   Verteiler_O2.Values[106] := 0.0;
   Verteiler_O2.Values[107] := 0.0;
   Verteiler_O2.Values[108] := 0.0;
   Verteiler_O2.Values[109] := 0.0;
   Verteiler_O2.Values[110] := 0.0;
   Verteiler_O2.Values[111] := 0.0;
   Verteiler_O2.Values[112] := 0.0;
   Verteiler_O2.Values[113] := 0.0;
   Verteiler_O2.Values[114] := 0.0;
   Verteiler_O2.Values[115] := 0.0;
   Verteiler_O2.Values[116] := 0.0;
   Verteiler_O2.Values[117] := 0.0;
   Verteiler_O2.Values[118] := 0.0;
   Verteiler_O2.Values[119] := 0.0;
   Verteiler_Temp.Values[0] := 0.0;
   Verteiler_Temp.Values[1] := 0.0;
   Verteiler_Temp.Values[2] := 0.0;
   Verteiler_Temp.Values[3] := 0.0;
   Verteiler_Temp.Values[4] := 0.0;
   Verteiler_Temp.Values[5] := 0.0;
   Verteiler_Temp.Values[6] := 0.0;
   Verteiler_Temp.Values[7] := 0.0;
   Verteiler_Temp.Values[8] := 0.0;
   Verteiler_Temp.Values[9] := 0.0;
   Verteiler_Temp.Values[10] := 0.0;
   Verteiler_Temp.Values[11] := 0.0;
   Verteiler_Temp.Values[12] := 0.0;
   Verteiler_Temp.Values[13] := 0.0;
   Verteiler_Temp.Values[14] := 0.0;
   Verteiler_Temp.Values[15] := 0.0;
   Verteiler_Temp.Values[16] := 0.0;
   Verteiler_Temp.Values[17] := 0.0;
   Verteiler_Temp.Values[18] := 0.0;
   Verteiler_Temp.Values[19] := 0.0;
   Verteiler_Temp.Values[20] := 0.0;
   Verteiler_Temp.Values[21] := 0.0;
   Verteiler_Temp.Values[22] := 0.0;
   Verteiler_Temp.Values[23] := 0.0;
   Verteiler_Temp.Values[24] := 0.0;
   Verteiler_Temp.Values[25] := 0.0;
   Verteiler_Temp.Values[26] := 0.0;
   Verteiler_Temp.Values[27] := 0.0;
   Verteiler_Temp.Values[28] := 0.0;
   Verteiler_Temp.Values[29] := 0.0;
   Verteiler_Temp.Values[30] := 0.0;
   Verteiler_Temp.Values[31] := 0.0;
   Verteiler_Temp.Values[32] := 0.0;
   Verteiler_Temp.Values[33] := 0.0;
   Verteiler_Temp.Values[34] := 0.0;
   Verteiler_Temp.Values[35] := 0.0;
   Verteiler_Temp.Values[36] := 0.0;
   Verteiler_Temp.Values[37] := 0.0;
   Verteiler_Temp.Values[38] := 0.0;
   Verteiler_Temp.Values[39] := 0.0;
   Verteiler_Temp.Values[40] := 0.0;
   Verteiler_Temp.Values[41] := 0.0;
   Verteiler_Temp.Values[42] := 0.0;
   Verteiler_Temp.Values[43] := 0.0;
   Verteiler_Temp.Values[44] := 0.0;
   Verteiler_Temp.Values[45] := 0.0;
   Verteiler_Temp.Values[46] := 0.0;
   Verteiler_Temp.Values[47] := 0.0;
   Verteiler_Temp.Values[48] := 0.0;
   Verteiler_Temp.Values[49] := 0.0;
   Verteiler_Temp.Values[50] := 0.0;
   Verteiler_Temp.Values[51] := 0.0;
   Verteiler_Temp.Values[52] := 0.0;
   Verteiler_Temp.Values[53] := 0.0;
   Verteiler_Temp.Values[54] := 0.0;
   Verteiler_Temp.Values[55] := 0.0;
   Verteiler_Temp.Values[56] := 0.0;
   Verteiler_Temp.Values[57] := 0.0;
   Verteiler_Temp.Values[58] := 0.0;
   Verteiler_Temp.Values[59] := 0.0;
   Verteiler_Temp.Values[60] := 0.0;
   Verteiler_Temp.Values[61] := 0.0;
   Verteiler_Temp.Values[62] := 0.0;
   Verteiler_Temp.Values[63] := 0.0;
   Verteiler_Temp.Values[64] := 0.0;
   Verteiler_Temp.Values[65] := 0.0;
   Verteiler_Temp.Values[66] := 0.0;
   Verteiler_Temp.Values[67] := 0.0;
   Verteiler_Temp.Values[68] := 0.0;
   Verteiler_Temp.Values[69] := 0.0;
   Verteiler_Temp.Values[70] := 0.0;
   Verteiler_Temp.Values[71] := 0.0;
   Verteiler_Temp.Values[72] := 0.0;
   Verteiler_Temp.Values[73] := 0.0;
   Verteiler_Temp.Values[74] := 0.0;
   Verteiler_Temp.Values[75] := 0.0;
   Verteiler_Temp.Values[76] := 0.0;
   Verteiler_Temp.Values[77] := 0.0;
   Verteiler_Temp.Values[78] := 0.0;
   Verteiler_Temp.Values[79] := 0.0;
   Verteiler_Temp.Values[80] := 0.0;
   Verteiler_Temp.Values[81] := 0.0;
   Verteiler_Temp.Values[82] := 0.0;
   Verteiler_Temp.Values[83] := 0.0;
   Verteiler_Temp.Values[84] := 0.0;
   Verteiler_Temp.Values[85] := 0.0;
   Verteiler_Temp.Values[86] := 0.0;
   Verteiler_Temp.Values[87] := 0.0;
   Verteiler_Temp.Values[88] := 0.0;
   Verteiler_Temp.Values[89] := 0.0;
   Verteiler_Temp.Values[90] := 0.0;
   Verteiler_Temp.Values[91] := 0.0;
   Verteiler_Temp.Values[92] := 0.0;
   Verteiler_Temp.Values[93] := 0.0;
   Verteiler_Temp.Values[94] := 0.0;
   Verteiler_Temp.Values[95] := 0.0;
   Verteiler_Temp.Values[96] := 0.0;
   Verteiler_Temp.Values[97] := 0.0;
   Verteiler_Temp.Values[98] := 0.0;
   Verteiler_Temp.Values[99] := 0.0;
   Verteiler_Temp.Values[100] := 0.0;
   Verteiler_Temp.Values[101] := 0.0;
   Verteiler_Temp.Values[102] := 0.0;
   Verteiler_Temp.Values[103] := 0.0;
   Verteiler_Temp.Values[104] := 0.0;
   Verteiler_Temp.Values[105] := 0.0;
   Verteiler_Temp.Values[106] := 0.0;
   Verteiler_Temp.Values[107] := 0.0;
   Verteiler_Temp.Values[108] := 0.0;
   Verteiler_Temp.Values[109] := 0.0;
   Verteiler_Temp.Values[110] := 0.0;
   Verteiler_Temp.Values[111] := 0.0;
   Verteiler_Temp.Values[112] := 0.0;
   Verteiler_Temp.Values[113] := 0.0;
   Verteiler_Temp.Values[114] := 0.0;
   Verteiler_Temp.Values[115] := 0.0;
   Verteiler_Temp.Values[116] := 0.0;
   Verteiler_Temp.Values[117] := 0.0;
   Verteiler_Temp.Values[118] := 0.0;
   Verteiler_Temp.Values[119] := 0.0;
   BB_UeSS_DF.Values[0] := -0.0063294;
   BB_UeSS_DF.Values[1] := -0.0063294;
   BB_UeSS_DF.Values[2] := -0.0063294;
   BB_UeSS_DF.Values[3] := -0.0063294;
   BB_UeSS_DF.Values[4] := -0.0063294;
   BB_UeSS_DF.Values[5] := -0.0063294;
   BB_UeSS_DF.Values[6] := -0.0063294;
   BB_UeSS_DF.Values[7] := -0.0063294;
   BB_UeSS_DF.Values[8] := -0.0099462;
   BB_UeSS_DF.Values[9] := -0.009042;
   BB_UeSS_DF.Values[10] := 0.0;
   BB_UeSS_DF.Values[11] := 0.0;
   BB_UeSS_DF.Values[12] := 0.0;
   BB_UeSS_DF.Values[13] := 0.0;
   BB_UeSS_DF.Values[14] := 0.0;
   BB_UeSS_DF.Values[15] := 0.0;
   BB_UeSS_DF.Values[16] := 0.0;
   BB_UeSS_DF.Values[17] := 0.0;
   BB_UeSS_DF.Values[18] := 0.0;
   BB_UeSS_DF.Values[19] := 0.0;
   BB_UeSS_DF.Values[20] := 0.0;
   BB_UeSS_DF.Values[21] := 0.0;
   BB_UeSS_DF.Values[22] := 0.0;
   BB_UeSS_DF.Values[23] := 0.0;
   BB_UeSS_DF.Values[24] := 0.0;
   BB_UeSS_DF.Values[25] := 0.0;
   BB_UeSS_DF.Values[26] := 0.0;
   BB_UeSS_DF.Values[27] := 0.0;
   BB_UeSS_DF.Values[28] := 0.0;
   BB_UeSS_DF.Values[29] := 0.0;
   BB_UeSS_DF.Values[30] := 0.0;
   BB_UeSS_DF.Values[31] := 0.0;
   BB_UeSS_DF.Values[32] := 0.0;
   BB_UeSS_DF.Values[33] := 0.0;
   BB_UeSS_DF.Values[34] := 0.0;
   BB_UeSS_DF.Values[35] := 0.0;
   BB_UeSS_DF.Values[36] := 0.0;
   BB_UeSS_DF.Values[37] := 0.0;
   BB_UeSS_DF.Values[38] := 0.0;
   BB_UeSS_DF.Values[39] := 0.0;
   BB_UeSS_DF.Values[40] := 0.0;
   BB_UeSS_DF.Values[41] := 0.0;
   BB_UeSS_DF.Values[42] := 0.0;
   BB_UeSS_DF.Values[43] := 0.0;
   BB_UeSS_DF.Values[44] := 0.0;
   BB_UeSS_DF.Values[45] := 0.0;
   BB_UeSS_DF.Values[46] := 0.0;
   BB_UeSS_DF.Values[47] := 0.0;
   BB_UeSS_DF.Values[48] := 0.0;
   BB_UeSS_DF.Values[49] := 0.0;
   BB_UeSS_DF.Values[50] := 0.0;
   BB_UeSS_DF.Values[51] := 0.0;
   BB_UeSS_DF.Values[52] := 0.0;
   BB_UeSS_DF.Values[53] := 0.0;
   BB_UeSS_DF.Values[54] := 0.0;
   BB_UeSS_DF.Values[55] := 0.0;
   BB_UeSS_DF.Values[56] := 0.0;
   BB_UeSS_DF.Values[57] := 0.0;
   BB_UeSS_DF.Values[58] := 0.0;
   BB_UeSS_DF.Values[59] := 0.0;
   BB_UeSS_DF.Values[60] := 0.0;
   BB_UeSS_DF.Values[61] := 0.0;
   BB_UeSS_DF.Values[62] := 0.0;
   BB_UeSS_DF.Values[63] := 0.0;
   BB_UeSS_DF.Values[64] := 0.0;
   BB_UeSS_DF.Values[65] := 0.0;
   BB_UeSS_DF.Values[66] := 0.0;
   BB_UeSS_DF.Values[67] := 0.0;
   BB_UeSS_DF.Values[68] := 0.0;
   BB_UeSS_DF.Values[69] := 0.0;
   BB_UeSS_DF.Values[70] := 0.0;
   BB_UeSS_DF.Values[71] := 0.0;
   BB_UeSS_DF.Values[72] := 0.0;
   BB_UeSS_DF.Values[73] := 0.0;
   BB_UeSS_DF.Values[74] := 0.0;
   BB_UeSS_DF.Values[75] := 0.0;
   BB_UeSS_DF.Values[76] := 0.0;
   BB_UeSS_DF.Values[77] := 0.0;
   BB_UeSS_DF.Values[78] := 0.0;
   BB_UeSS_DF.Values[79] := 0.0;
   BB_UeSS_DF.Values[80] := 0.0;
   BB_UeSS_DF.Values[81] := 0.0;
   BB_UeSS_DF.Values[82] := 0.0;
   BB_UeSS_DF.Values[83] := 0.0;
   BB_UeSS_DF.Values[84] := 0.0;
   BB_UeSS_DF.Values[85] := 0.0;
   BB_UeSS_DF.Values[86] := 0.0;
   BB_UeSS_DF.Values[87] := 0.0;
   BB_UeSS_DF.Values[88] := 0.0;
   BB_UeSS_DF.Values[89] := 0.0;
   BB_UeSS_DF.Values[90] := 0.0;
   BB_UeSS_DF.Values[91] := 0.0;
   BB_UeSS_DF.Values[92] := 0.0;
   BB_UeSS_DF.Values[93] := 0.0;
   BB_UeSS_DF.Values[94] := 0.0;
   BB_UeSS_DF.Values[95] := 0.0;
   BB_UeSS_DF.Values[96] := 0.0;
   BB_UeSS_DF.Values[97] := 0.0;
   BB_UeSS_DF.Values[98] := 0.0;
   BB_UeSS_DF.Values[99] := 0.0;
   BB_UeSS_DF.Values[100] := 0.0;
   BB_UeSS_DF.Values[101] := 0.0;
   BB_UeSS_DF.Values[102] := 0.0;
   BB_UeSS_DF.Values[103] := 0.0;
   BB_UeSS_DF.Values[104] := 0.0;
   BB_UeSS_DF.Values[105] := 0.0;
   BB_UeSS_DF.Values[106] := 0.0;
   BB_UeSS_DF.Values[107] := 0.0;
   BB_UeSS_DF.Values[108] := 0.0;
   BB_UeSS_DF.Values[109] := 0.0;
   BB_UeSS_DF.Values[110] := 0.0;
   BB_UeSS_DF.Values[111] := 0.0;
   BB_UeSS_DF.Values[112] := 0.0;
   BB_UeSS_DF.Values[113] := 0.0;
   BB_UeSS_DF.Values[114] := 0.0;
   BB_UeSS_DF.Values[115] := 0.0;
   BB_UeSS_DF.Values[116] := 0.0;
   BB_UeSS_DF.Values[117] := 0.0;
   BB_UeSS_DF.Values[118] := 0.0;
   BB_UeSS_DF.Values[119] := 0.0;
   Ablauf_DF.Values[0] := 11.22745;
   Ablauf_DF.Values[1] := 11.21796;
   Ablauf_DF.Values[2] := 11.20439;
   Ablauf_DF.Values[3] := 11.19897;
   Ablauf_DF.Values[4] := 11.18948;
   Ablauf_DF.Values[5] := 11.18541;
   Ablauf_DF.Values[6] := 11.1949;
   Ablauf_DF.Values[7] := 11.22338;
   Ablauf_DF.Values[8] := 11.2383;
   Ablauf_DF.Values[9] := 11.22745;
   Ablauf_DF.Values[10] := 0.0;
   Ablauf_DF.Values[11] := 0.0;
   Ablauf_DF.Values[12] := 0.0;
   Ablauf_DF.Values[13] := 0.0;
   Ablauf_DF.Values[14] := 0.0;
   Ablauf_DF.Values[15] := 0.0;
   Ablauf_DF.Values[16] := 0.0;
   Ablauf_DF.Values[17] := 0.0;
   Ablauf_DF.Values[18] := 0.0;
   Ablauf_DF.Values[19] := 0.0;
   Ablauf_DF.Values[20] := 0.0;
   Ablauf_DF.Values[21] := 0.0;
   Ablauf_DF.Values[22] := 0.0;
   Ablauf_DF.Values[23] := 0.0;
   Ablauf_DF.Values[24] := 0.0;
   Ablauf_DF.Values[25] := 0.0;
   Ablauf_DF.Values[26] := 0.0;
   Ablauf_DF.Values[27] := 0.0;
   Ablauf_DF.Values[28] := 0.0;
   Ablauf_DF.Values[29] := 0.0;
   Ablauf_DF.Values[30] := 0.0;
   Ablauf_DF.Values[31] := 0.0;
   Ablauf_DF.Values[32] := 0.0;
   Ablauf_DF.Values[33] := 0.0;
   Ablauf_DF.Values[34] := 0.0;
   Ablauf_DF.Values[35] := 0.0;
   Ablauf_DF.Values[36] := 0.0;
   Ablauf_DF.Values[37] := 0.0;
   Ablauf_DF.Values[38] := 0.0;
   Ablauf_DF.Values[39] := 0.0;
   Ablauf_DF.Values[40] := 0.0;
   Ablauf_DF.Values[41] := 0.0;
   Ablauf_DF.Values[42] := 0.0;
   Ablauf_DF.Values[43] := 0.0;
   Ablauf_DF.Values[44] := 0.0;
   Ablauf_DF.Values[45] := 0.0;
   Ablauf_DF.Values[46] := 0.0;
   Ablauf_DF.Values[47] := 0.0;
   Ablauf_DF.Values[48] := 0.0;
   Ablauf_DF.Values[49] := 0.0;
   Ablauf_DF.Values[50] := 0.0;
   Ablauf_DF.Values[51] := 0.0;
   Ablauf_DF.Values[52] := 0.0;
   Ablauf_DF.Values[53] := 0.0;
   Ablauf_DF.Values[54] := 0.0;
   Ablauf_DF.Values[55] := 0.0;
   Ablauf_DF.Values[56] := 0.0;
   Ablauf_DF.Values[57] := 0.0;
   Ablauf_DF.Values[58] := 0.0;
   Ablauf_DF.Values[59] := 0.0;
   Ablauf_DF.Values[60] := 0.0;
   Ablauf_DF.Values[61] := 0.0;
   Ablauf_DF.Values[62] := 0.0;
   Ablauf_DF.Values[63] := 0.0;
   Ablauf_DF.Values[64] := 0.0;
   Ablauf_DF.Values[65] := 0.0;
   Ablauf_DF.Values[66] := 0.0;
   Ablauf_DF.Values[67] := 0.0;
   Ablauf_DF.Values[68] := 0.0;
   Ablauf_DF.Values[69] := 0.0;
   Ablauf_DF.Values[70] := 0.0;
   Ablauf_DF.Values[71] := 0.0;
   Ablauf_DF.Values[72] := 0.0;
   Ablauf_DF.Values[73] := 0.0;
   Ablauf_DF.Values[74] := 0.0;
   Ablauf_DF.Values[75] := 0.0;
   Ablauf_DF.Values[76] := 0.0;
   Ablauf_DF.Values[77] := 0.0;
   Ablauf_DF.Values[78] := 0.0;
   Ablauf_DF.Values[79] := 0.0;
   Ablauf_DF.Values[80] := 0.0;
   Ablauf_DF.Values[81] := 0.0;
   Ablauf_DF.Values[82] := 0.0;
   Ablauf_DF.Values[83] := 0.0;
   Ablauf_DF.Values[84] := 0.0;
   Ablauf_DF.Values[85] := 0.0;
   Ablauf_DF.Values[86] := 0.0;
   Ablauf_DF.Values[87] := 0.0;
   Ablauf_DF.Values[88] := 0.0;
   Ablauf_DF.Values[89] := 0.0;
   Ablauf_DF.Values[90] := 0.0;
   Ablauf_DF.Values[91] := 0.0;
   Ablauf_DF.Values[92] := 0.0;
   Ablauf_DF.Values[93] := 0.0;
   Ablauf_DF.Values[94] := 0.0;
   Ablauf_DF.Values[95] := 0.0;
   Ablauf_DF.Values[96] := 0.0;
   Ablauf_DF.Values[97] := 0.0;
   Ablauf_DF.Values[98] := 0.0;
   Ablauf_DF.Values[99] := 0.0;
   Ablauf_DF.Values[100] := 0.0;
   Ablauf_DF.Values[101] := 0.0;
   Ablauf_DF.Values[102] := 0.0;
   Ablauf_DF.Values[103] := 0.0;
   Ablauf_DF.Values[104] := 0.0;
   Ablauf_DF.Values[105] := 0.0;
   Ablauf_DF.Values[106] := 0.0;
   Ablauf_DF.Values[107] := 0.0;
   Ablauf_DF.Values[108] := 0.0;
   Ablauf_DF.Values[109] := 0.0;
   Ablauf_DF.Values[110] := 0.0;
   Ablauf_DF.Values[111] := 0.0;
   Ablauf_DF.Values[112] := 0.0;
   Ablauf_DF.Values[113] := 0.0;
   Ablauf_DF.Values[114] := 0.0;
   Ablauf_DF.Values[115] := 0.0;
   Ablauf_DF.Values[116] := 0.0;
   Ablauf_DF.Values[117] := 0.0;
   Ablauf_DF.Values[118] := 0.0;
   Ablauf_DF.Values[119] := 0.0;
   Ablauf_pH.Values[0] := 7.047787;
   Ablauf_pH.Values[1] := 7.047787;
   Ablauf_pH.Values[2] := 7.047787;
   Ablauf_pH.Values[3] := 7.047787;
   Ablauf_pH.Values[4] := 7.047787;
   Ablauf_pH.Values[5] := 7.047787;
   Ablauf_pH.Values[6] := 7.047787;
   Ablauf_pH.Values[7] := 7.047787;
   Ablauf_pH.Values[8] := 7.047787;
   Ablauf_pH.Values[9] := 7.047787;
   Ablauf_pH.Values[10] := 0.0;
   Ablauf_pH.Values[11] := 0.0;
   Ablauf_pH.Values[12] := 0.0;
   Ablauf_pH.Values[13] := 0.0;
   Ablauf_pH.Values[14] := 0.0;
   Ablauf_pH.Values[15] := 0.0;
   Ablauf_pH.Values[16] := 0.0;
   Ablauf_pH.Values[17] := 0.0;
   Ablauf_pH.Values[18] := 0.0;
   Ablauf_pH.Values[19] := 0.0;
   Ablauf_pH.Values[20] := 0.0;
   Ablauf_pH.Values[21] := 0.0;
   Ablauf_pH.Values[22] := 0.0;
   Ablauf_pH.Values[23] := 0.0;
   Ablauf_pH.Values[24] := 0.0;
   Ablauf_pH.Values[25] := 0.0;
   Ablauf_pH.Values[26] := 0.0;
   Ablauf_pH.Values[27] := 0.0;
   Ablauf_pH.Values[28] := 0.0;
   Ablauf_pH.Values[29] := 0.0;
   Ablauf_pH.Values[30] := 0.0;
   Ablauf_pH.Values[31] := 0.0;
   Ablauf_pH.Values[32] := 0.0;
   Ablauf_pH.Values[33] := 0.0;
   Ablauf_pH.Values[34] := 0.0;
   Ablauf_pH.Values[35] := 0.0;
   Ablauf_pH.Values[36] := 0.0;
   Ablauf_pH.Values[37] := 0.0;
   Ablauf_pH.Values[38] := 0.0;
   Ablauf_pH.Values[39] := 0.0;
   Ablauf_pH.Values[40] := 0.0;
   Ablauf_pH.Values[41] := 0.0;
   Ablauf_pH.Values[42] := 0.0;
   Ablauf_pH.Values[43] := 0.0;
   Ablauf_pH.Values[44] := 0.0;
   Ablauf_pH.Values[45] := 0.0;
   Ablauf_pH.Values[46] := 0.0;
   Ablauf_pH.Values[47] := 0.0;
   Ablauf_pH.Values[48] := 0.0;
   Ablauf_pH.Values[49] := 0.0;
   Ablauf_pH.Values[50] := 0.0;
   Ablauf_pH.Values[51] := 0.0;
   Ablauf_pH.Values[52] := 0.0;
   Ablauf_pH.Values[53] := 0.0;
   Ablauf_pH.Values[54] := 0.0;
   Ablauf_pH.Values[55] := 0.0;
   Ablauf_pH.Values[56] := 0.0;
   Ablauf_pH.Values[57] := 0.0;
   Ablauf_pH.Values[58] := 0.0;
   Ablauf_pH.Values[59] := 0.0;
   Ablauf_pH.Values[60] := 0.0;
   Ablauf_pH.Values[61] := 0.0;
   Ablauf_pH.Values[62] := 0.0;
   Ablauf_pH.Values[63] := 0.0;
   Ablauf_pH.Values[64] := 0.0;
   Ablauf_pH.Values[65] := 0.0;
   Ablauf_pH.Values[66] := 0.0;
   Ablauf_pH.Values[67] := 0.0;
   Ablauf_pH.Values[68] := 0.0;
   Ablauf_pH.Values[69] := 0.0;
   Ablauf_pH.Values[70] := 0.0;
   Ablauf_pH.Values[71] := 0.0;
   Ablauf_pH.Values[72] := 0.0;
   Ablauf_pH.Values[73] := 0.0;
   Ablauf_pH.Values[74] := 0.0;
   Ablauf_pH.Values[75] := 0.0;
   Ablauf_pH.Values[76] := 0.0;
   Ablauf_pH.Values[77] := 0.0;
   Ablauf_pH.Values[78] := 0.0;
   Ablauf_pH.Values[79] := 0.0;
   Ablauf_pH.Values[80] := 0.0;
   Ablauf_pH.Values[81] := 0.0;
   Ablauf_pH.Values[82] := 0.0;
   Ablauf_pH.Values[83] := 0.0;
   Ablauf_pH.Values[84] := 0.0;
   Ablauf_pH.Values[85] := 0.0;
   Ablauf_pH.Values[86] := 0.0;
   Ablauf_pH.Values[87] := 0.0;
   Ablauf_pH.Values[88] := 0.0;
   Ablauf_pH.Values[89] := 0.0;
   Ablauf_pH.Values[90] := 0.0;
   Ablauf_pH.Values[91] := 0.0;
   Ablauf_pH.Values[92] := 0.0;
   Ablauf_pH.Values[93] := 0.0;
   Ablauf_pH.Values[94] := 0.0;
   Ablauf_pH.Values[95] := 0.0;
   Ablauf_pH.Values[96] := 0.0;
   Ablauf_pH.Values[97] := 0.0;
   Ablauf_pH.Values[98] := 0.0;
   Ablauf_pH.Values[99] := 0.0;
   Ablauf_pH.Values[100] := 0.0;
   Ablauf_pH.Values[101] := 0.0;
   Ablauf_pH.Values[102] := 0.0;
   Ablauf_pH.Values[103] := 0.0;
   Ablauf_pH.Values[104] := 0.0;
   Ablauf_pH.Values[105] := 0.0;
   Ablauf_pH.Values[106] := 0.0;
   Ablauf_pH.Values[107] := 0.0;
   Ablauf_pH.Values[108] := 0.0;
   Ablauf_pH.Values[109] := 0.0;
   Ablauf_pH.Values[110] := 0.0;
   Ablauf_pH.Values[111] := 0.0;
   Ablauf_pH.Values[112] := 0.0;
   Ablauf_pH.Values[113] := 0.0;
   Ablauf_pH.Values[114] := 0.0;
   Ablauf_pH.Values[115] := 0.0;
   Ablauf_pH.Values[116] := 0.0;
   Ablauf_pH.Values[117] := 0.0;
   Ablauf_pH.Values[118] := 0.0;
   Ablauf_pH.Values[119] := 0.0;
   Ablauf_O2.Values[0] := 1.460735;
   Ablauf_O2.Values[1] := 1.460735;
   Ablauf_O2.Values[2] := 1.460735;
   Ablauf_O2.Values[3] := 1.460735;
   Ablauf_O2.Values[4] := 1.460735;
   Ablauf_O2.Values[5] := 1.460735;
   Ablauf_O2.Values[6] := 1.460735;
   Ablauf_O2.Values[7] := 1.460735;
   Ablauf_O2.Values[8] := 1.460735;
   Ablauf_O2.Values[9] := 1.460735;
   Ablauf_O2.Values[10] := 0.0;
   Ablauf_O2.Values[11] := 0.0;
   Ablauf_O2.Values[12] := 0.0;
   Ablauf_O2.Values[13] := 0.0;
   Ablauf_O2.Values[14] := 0.0;
   Ablauf_O2.Values[15] := 0.0;
   Ablauf_O2.Values[16] := 0.0;
   Ablauf_O2.Values[17] := 0.0;
   Ablauf_O2.Values[18] := 0.0;
   Ablauf_O2.Values[19] := 0.0;
   Ablauf_O2.Values[20] := 0.0;
   Ablauf_O2.Values[21] := 0.0;
   Ablauf_O2.Values[22] := 0.0;
   Ablauf_O2.Values[23] := 0.0;
   Ablauf_O2.Values[24] := 0.0;
   Ablauf_O2.Values[25] := 0.0;
   Ablauf_O2.Values[26] := 0.0;
   Ablauf_O2.Values[27] := 0.0;
   Ablauf_O2.Values[28] := 0.0;
   Ablauf_O2.Values[29] := 0.0;
   Ablauf_O2.Values[30] := 0.0;
   Ablauf_O2.Values[31] := 0.0;
   Ablauf_O2.Values[32] := 0.0;
   Ablauf_O2.Values[33] := 0.0;
   Ablauf_O2.Values[34] := 0.0;
   Ablauf_O2.Values[35] := 0.0;
   Ablauf_O2.Values[36] := 0.0;
   Ablauf_O2.Values[37] := 0.0;
   Ablauf_O2.Values[38] := 0.0;
   Ablauf_O2.Values[39] := 0.0;
   Ablauf_O2.Values[40] := 0.0;
   Ablauf_O2.Values[41] := 0.0;
   Ablauf_O2.Values[42] := 0.0;
   Ablauf_O2.Values[43] := 0.0;
   Ablauf_O2.Values[44] := 0.0;
   Ablauf_O2.Values[45] := 0.0;
   Ablauf_O2.Values[46] := 0.0;
   Ablauf_O2.Values[47] := 0.0;
   Ablauf_O2.Values[48] := 0.0;
   Ablauf_O2.Values[49] := 0.0;
   Ablauf_O2.Values[50] := 0.0;
   Ablauf_O2.Values[51] := 0.0;
   Ablauf_O2.Values[52] := 0.0;
   Ablauf_O2.Values[53] := 0.0;
   Ablauf_O2.Values[54] := 0.0;
   Ablauf_O2.Values[55] := 0.0;
   Ablauf_O2.Values[56] := 0.0;
   Ablauf_O2.Values[57] := 0.0;
   Ablauf_O2.Values[58] := 0.0;
   Ablauf_O2.Values[59] := 0.0;
   Ablauf_O2.Values[60] := 0.0;
   Ablauf_O2.Values[61] := 0.0;
   Ablauf_O2.Values[62] := 0.0;
   Ablauf_O2.Values[63] := 0.0;
   Ablauf_O2.Values[64] := 0.0;
   Ablauf_O2.Values[65] := 0.0;
   Ablauf_O2.Values[66] := 0.0;
   Ablauf_O2.Values[67] := 0.0;
   Ablauf_O2.Values[68] := 0.0;
   Ablauf_O2.Values[69] := 0.0;
   Ablauf_O2.Values[70] := 0.0;
   Ablauf_O2.Values[71] := 0.0;
   Ablauf_O2.Values[72] := 0.0;
   Ablauf_O2.Values[73] := 0.0;
   Ablauf_O2.Values[74] := 0.0;
   Ablauf_O2.Values[75] := 0.0;
   Ablauf_O2.Values[76] := 0.0;
   Ablauf_O2.Values[77] := 0.0;
   Ablauf_O2.Values[78] := 0.0;
   Ablauf_O2.Values[79] := 0.0;
   Ablauf_O2.Values[80] := 0.0;
   Ablauf_O2.Values[81] := 0.0;
   Ablauf_O2.Values[82] := 0.0;
   Ablauf_O2.Values[83] := 0.0;
   Ablauf_O2.Values[84] := 0.0;
   Ablauf_O2.Values[85] := 0.0;
   Ablauf_O2.Values[86] := 0.0;
   Ablauf_O2.Values[87] := 0.0;
   Ablauf_O2.Values[88] := 0.0;
   Ablauf_O2.Values[89] := 0.0;
   Ablauf_O2.Values[90] := 0.0;
   Ablauf_O2.Values[91] := 0.0;
   Ablauf_O2.Values[92] := 0.0;
   Ablauf_O2.Values[93] := 0.0;
   Ablauf_O2.Values[94] := 0.0;
   Ablauf_O2.Values[95] := 0.0;
   Ablauf_O2.Values[96] := 0.0;
   Ablauf_O2.Values[97] := 0.0;
   Ablauf_O2.Values[98] := 0.0;
   Ablauf_O2.Values[99] := 0.0;
   Ablauf_O2.Values[100] := 0.0;
   Ablauf_O2.Values[101] := 0.0;
   Ablauf_O2.Values[102] := 0.0;
   Ablauf_O2.Values[103] := 0.0;
   Ablauf_O2.Values[104] := 0.0;
   Ablauf_O2.Values[105] := 0.0;
   Ablauf_O2.Values[106] := 0.0;
   Ablauf_O2.Values[107] := 0.0;
   Ablauf_O2.Values[108] := 0.0;
   Ablauf_O2.Values[109] := 0.0;
   Ablauf_O2.Values[110] := 0.0;
   Ablauf_O2.Values[111] := 0.0;
   Ablauf_O2.Values[112] := 0.0;
   Ablauf_O2.Values[113] := 0.0;
   Ablauf_O2.Values[114] := 0.0;
   Ablauf_O2.Values[115] := 0.0;
   Ablauf_O2.Values[116] := 0.0;
   Ablauf_O2.Values[117] := 0.0;
   Ablauf_O2.Values[118] := 0.0;
   Ablauf_O2.Values[119] := 0.0;
   Ablauf_Temp.Values[0] := 12.94814;
   Ablauf_Temp.Values[1] := 12.94588;
   Ablauf_Temp.Values[2] := 12.94588;
   Ablauf_Temp.Values[3] := 12.94588;
   Ablauf_Temp.Values[4] := 12.94588;
   Ablauf_Temp.Values[5] := 12.94814;
   Ablauf_Temp.Values[6] := 12.94814;
   Ablauf_Temp.Values[7] := 12.94588;
   Ablauf_Temp.Values[8] := 12.94588;
   Ablauf_Temp.Values[9] := 12.94814;
   Ablauf_Temp.Values[10] := 0.0;
   Ablauf_Temp.Values[11] := 0.0;
   Ablauf_Temp.Values[12] := 0.0;
   Ablauf_Temp.Values[13] := 0.0;
   Ablauf_Temp.Values[14] := 0.0;
   Ablauf_Temp.Values[15] := 0.0;
   Ablauf_Temp.Values[16] := 0.0;
   Ablauf_Temp.Values[17] := 0.0;
   Ablauf_Temp.Values[18] := 0.0;
   Ablauf_Temp.Values[19] := 0.0;
   Ablauf_Temp.Values[20] := 0.0;
   Ablauf_Temp.Values[21] := 0.0;
   Ablauf_Temp.Values[22] := 0.0;
   Ablauf_Temp.Values[23] := 0.0;
   Ablauf_Temp.Values[24] := 0.0;
   Ablauf_Temp.Values[25] := 0.0;
   Ablauf_Temp.Values[26] := 0.0;
   Ablauf_Temp.Values[27] := 0.0;
   Ablauf_Temp.Values[28] := 0.0;
   Ablauf_Temp.Values[29] := 0.0;
   Ablauf_Temp.Values[30] := 0.0;
   Ablauf_Temp.Values[31] := 0.0;
   Ablauf_Temp.Values[32] := 0.0;
   Ablauf_Temp.Values[33] := 0.0;
   Ablauf_Temp.Values[34] := 0.0;
   Ablauf_Temp.Values[35] := 0.0;
   Ablauf_Temp.Values[36] := 0.0;
   Ablauf_Temp.Values[37] := 0.0;
   Ablauf_Temp.Values[38] := 0.0;
   Ablauf_Temp.Values[39] := 0.0;
   Ablauf_Temp.Values[40] := 0.0;
   Ablauf_Temp.Values[41] := 0.0;
   Ablauf_Temp.Values[42] := 0.0;
   Ablauf_Temp.Values[43] := 0.0;
   Ablauf_Temp.Values[44] := 0.0;
   Ablauf_Temp.Values[45] := 0.0;
   Ablauf_Temp.Values[46] := 0.0;
   Ablauf_Temp.Values[47] := 0.0;
   Ablauf_Temp.Values[48] := 0.0;
   Ablauf_Temp.Values[49] := 0.0;
   Ablauf_Temp.Values[50] := 0.0;
   Ablauf_Temp.Values[51] := 0.0;
   Ablauf_Temp.Values[52] := 0.0;
   Ablauf_Temp.Values[53] := 0.0;
   Ablauf_Temp.Values[54] := 0.0;
   Ablauf_Temp.Values[55] := 0.0;
   Ablauf_Temp.Values[56] := 0.0;
   Ablauf_Temp.Values[57] := 0.0;
   Ablauf_Temp.Values[58] := 0.0;
   Ablauf_Temp.Values[59] := 0.0;
   Ablauf_Temp.Values[60] := 0.0;
   Ablauf_Temp.Values[61] := 0.0;
   Ablauf_Temp.Values[62] := 0.0;
   Ablauf_Temp.Values[63] := 0.0;
   Ablauf_Temp.Values[64] := 0.0;
   Ablauf_Temp.Values[65] := 0.0;
   Ablauf_Temp.Values[66] := 0.0;
   Ablauf_Temp.Values[67] := 0.0;
   Ablauf_Temp.Values[68] := 0.0;
   Ablauf_Temp.Values[69] := 0.0;
   Ablauf_Temp.Values[70] := 0.0;
   Ablauf_Temp.Values[71] := 0.0;
   Ablauf_Temp.Values[72] := 0.0;
   Ablauf_Temp.Values[73] := 0.0;
   Ablauf_Temp.Values[74] := 0.0;
   Ablauf_Temp.Values[75] := 0.0;
   Ablauf_Temp.Values[76] := 0.0;
   Ablauf_Temp.Values[77] := 0.0;
   Ablauf_Temp.Values[78] := 0.0;
   Ablauf_Temp.Values[79] := 0.0;
   Ablauf_Temp.Values[80] := 0.0;
   Ablauf_Temp.Values[81] := 0.0;
   Ablauf_Temp.Values[82] := 0.0;
   Ablauf_Temp.Values[83] := 0.0;
   Ablauf_Temp.Values[84] := 0.0;
   Ablauf_Temp.Values[85] := 0.0;
   Ablauf_Temp.Values[86] := 0.0;
   Ablauf_Temp.Values[87] := 0.0;
   Ablauf_Temp.Values[88] := 0.0;
   Ablauf_Temp.Values[89] := 0.0;
   Ablauf_Temp.Values[90] := 0.0;
   Ablauf_Temp.Values[91] := 0.0;
   Ablauf_Temp.Values[92] := 0.0;
   Ablauf_Temp.Values[93] := 0.0;
   Ablauf_Temp.Values[94] := 0.0;
   Ablauf_Temp.Values[95] := 0.0;
   Ablauf_Temp.Values[96] := 0.0;
   Ablauf_Temp.Values[97] := 0.0;
   Ablauf_Temp.Values[98] := 0.0;
   Ablauf_Temp.Values[99] := 0.0;
   Ablauf_Temp.Values[100] := 0.0;
   Ablauf_Temp.Values[101] := 0.0;
   Ablauf_Temp.Values[102] := 0.0;
   Ablauf_Temp.Values[103] := 0.0;
   Ablauf_Temp.Values[104] := 0.0;
   Ablauf_Temp.Values[105] := 0.0;
   Ablauf_Temp.Values[106] := 0.0;
   Ablauf_Temp.Values[107] := 0.0;
   Ablauf_Temp.Values[108] := 0.0;
   Ablauf_Temp.Values[109] := 0.0;
   Ablauf_Temp.Values[110] := 0.0;
   Ablauf_Temp.Values[111] := 0.0;
   Ablauf_Temp.Values[112] := 0.0;
   Ablauf_Temp.Values[113] := 0.0;
   Ablauf_Temp.Values[114] := 0.0;
   Ablauf_Temp.Values[115] := 0.0;
   Ablauf_Temp.Values[116] := 0.0;
   Ablauf_Temp.Values[117] := 0.0;
   Ablauf_Temp.Values[118] := 0.0;
   Ablauf_Temp.Values[119] := 0.0;
   Schlamm_ED_Niv.Values[0] := 0.0;
   Schlamm_ED_Niv.Values[1] := 0.0;
   Schlamm_ED_Niv.Values[2] := 0.0;
   Schlamm_ED_Niv.Values[3] := 0.0;
   Schlamm_ED_Niv.Values[4] := 0.0;
   Schlamm_ED_Niv.Values[5] := 0.0;
   Schlamm_ED_Niv.Values[6] := 0.0;
   Schlamm_ED_Niv.Values[7] := 0.0;
   Schlamm_ED_Niv.Values[8] := 0.0;
   Schlamm_ED_Niv.Values[9] := 0.0;
   Schlamm_ED_Niv.Values[10] := 0.0;
   Schlamm_ED_Niv.Values[11] := 0.0;
   Schlamm_ED_Niv.Values[12] := 0.0;
   Schlamm_ED_Niv.Values[13] := 0.0;
   Schlamm_ED_Niv.Values[14] := 0.0;
   Schlamm_ED_Niv.Values[15] := 0.0;
   Schlamm_ED_Niv.Values[16] := 0.0;
   Schlamm_ED_Niv.Values[17] := 0.0;
   Schlamm_ED_Niv.Values[18] := 0.0;
   Schlamm_ED_Niv.Values[19] := 0.0;
   Schlamm_ED_Niv.Values[20] := 0.0;
   Schlamm_ED_Niv.Values[21] := 0.0;
   Schlamm_ED_Niv.Values[22] := 0.0;
   Schlamm_ED_Niv.Values[23] := 0.0;
   Schlamm_ED_Niv.Values[24] := 0.0;
   Schlamm_ED_Niv.Values[25] := 0.0;
   Schlamm_ED_Niv.Values[26] := 0.0;
   Schlamm_ED_Niv.Values[27] := 0.0;
   Schlamm_ED_Niv.Values[28] := 0.0;
   Schlamm_ED_Niv.Values[29] := 0.0;
   Schlamm_ED_Niv.Values[30] := 0.0;
   Schlamm_ED_Niv.Values[31] := 0.0;
   Schlamm_ED_Niv.Values[32] := 0.0;
   Schlamm_ED_Niv.Values[33] := 0.0;
   Schlamm_ED_Niv.Values[34] := 0.0;
   Schlamm_ED_Niv.Values[35] := 0.0;
   Schlamm_ED_Niv.Values[36] := 0.0;
   Schlamm_ED_Niv.Values[37] := 0.0;
   Schlamm_ED_Niv.Values[38] := 0.0;
   Schlamm_ED_Niv.Values[39] := 0.0;
   Schlamm_ED_Niv.Values[40] := 0.0;
   Schlamm_ED_Niv.Values[41] := 0.0;
   Schlamm_ED_Niv.Values[42] := 0.0;
   Schlamm_ED_Niv.Values[43] := 0.0;
   Schlamm_ED_Niv.Values[44] := 0.0;
   Schlamm_ED_Niv.Values[45] := 0.0;
   Schlamm_ED_Niv.Values[46] := 0.0;
   Schlamm_ED_Niv.Values[47] := 0.0;
   Schlamm_ED_Niv.Values[48] := 0.0;
   Schlamm_ED_Niv.Values[49] := 0.0;
   Schlamm_ED_Niv.Values[50] := 0.0;
   Schlamm_ED_Niv.Values[51] := 0.0;
   Schlamm_ED_Niv.Values[52] := 0.0;
   Schlamm_ED_Niv.Values[53] := 0.0;
   Schlamm_ED_Niv.Values[54] := 0.0;
   Schlamm_ED_Niv.Values[55] := 0.0;
   Schlamm_ED_Niv.Values[56] := 0.0;
   Schlamm_ED_Niv.Values[57] := 0.0;
   Schlamm_ED_Niv.Values[58] := 0.0;
   Schlamm_ED_Niv.Values[59] := 0.0;
   Schlamm_ED_Niv.Values[60] := 0.0;
   Schlamm_ED_Niv.Values[61] := 0.0;
   Schlamm_ED_Niv.Values[62] := 0.0;
   Schlamm_ED_Niv.Values[63] := 0.0;
   Schlamm_ED_Niv.Values[64] := 0.0;
   Schlamm_ED_Niv.Values[65] := 0.0;
   Schlamm_ED_Niv.Values[66] := 0.0;
   Schlamm_ED_Niv.Values[67] := 0.0;
   Schlamm_ED_Niv.Values[68] := 0.0;
   Schlamm_ED_Niv.Values[69] := 0.0;
   Schlamm_ED_Niv.Values[70] := 0.0;
   Schlamm_ED_Niv.Values[71] := 0.0;
   Schlamm_ED_Niv.Values[72] := 0.0;
   Schlamm_ED_Niv.Values[73] := 0.0;
   Schlamm_ED_Niv.Values[74] := 0.0;
   Schlamm_ED_Niv.Values[75] := 0.0;
   Schlamm_ED_Niv.Values[76] := 0.0;
   Schlamm_ED_Niv.Values[77] := 0.0;
   Schlamm_ED_Niv.Values[78] := 0.0;
   Schlamm_ED_Niv.Values[79] := 0.0;
   Schlamm_ED_Niv.Values[80] := 0.0;
   Schlamm_ED_Niv.Values[81] := 0.0;
   Schlamm_ED_Niv.Values[82] := 0.0;
   Schlamm_ED_Niv.Values[83] := 0.0;
   Schlamm_ED_Niv.Values[84] := 0.0;
   Schlamm_ED_Niv.Values[85] := 0.0;
   Schlamm_ED_Niv.Values[86] := 0.0;
   Schlamm_ED_Niv.Values[87] := 0.0;
   Schlamm_ED_Niv.Values[88] := 0.0;
   Schlamm_ED_Niv.Values[89] := 0.0;
   Schlamm_ED_Niv.Values[90] := 0.0;
   Schlamm_ED_Niv.Values[91] := 0.0;
   Schlamm_ED_Niv.Values[92] := 0.0;
   Schlamm_ED_Niv.Values[93] := 0.0;
   Schlamm_ED_Niv.Values[94] := 0.0;
   Schlamm_ED_Niv.Values[95] := 0.0;
   Schlamm_ED_Niv.Values[96] := 0.0;
   Schlamm_ED_Niv.Values[97] := 0.0;
   Schlamm_ED_Niv.Values[98] := 0.0;
   Schlamm_ED_Niv.Values[99] := 0.0;
   Schlamm_ED_Niv.Values[100] := 0.0;
   Schlamm_ED_Niv.Values[101] := 0.0;
   Schlamm_ED_Niv.Values[102] := 0.0;
   Schlamm_ED_Niv.Values[103] := 0.0;
   Schlamm_ED_Niv.Values[104] := 0.0;
   Schlamm_ED_Niv.Values[105] := 0.0;
   Schlamm_ED_Niv.Values[106] := 0.0;
   Schlamm_ED_Niv.Values[107] := 0.0;
   Schlamm_ED_Niv.Values[108] := 0.0;
   Schlamm_ED_Niv.Values[109] := 0.0;
   Schlamm_ED_Niv.Values[110] := 0.0;
   Schlamm_ED_Niv.Values[111] := 0.0;
   Schlamm_ED_Niv.Values[112] := 0.0;
   Schlamm_ED_Niv.Values[113] := 0.0;
   Schlamm_ED_Niv.Values[114] := 0.0;
   Schlamm_ED_Niv.Values[115] := 0.0;
   Schlamm_ED_Niv.Values[116] := 0.0;
   Schlamm_ED_Niv.Values[117] := 0.0;
   Schlamm_ED_Niv.Values[118] := 0.0;
   Schlamm_ED_Niv.Values[119] := 0.0;
   Schlamm_Besch_Niv.Values[0] := 0.0;
   Schlamm_Besch_Niv.Values[1] := 0.0;
   Schlamm_Besch_Niv.Values[2] := 0.0;
   Schlamm_Besch_Niv.Values[3] := 0.0;
   Schlamm_Besch_Niv.Values[4] := 0.0;
   Schlamm_Besch_Niv.Values[5] := 0.0;
   Schlamm_Besch_Niv.Values[6] := 0.0;
   Schlamm_Besch_Niv.Values[7] := 0.0;
   Schlamm_Besch_Niv.Values[8] := 0.0;
   Schlamm_Besch_Niv.Values[9] := 0.0;
   Schlamm_Besch_Niv.Values[10] := 0.0;
   Schlamm_Besch_Niv.Values[11] := 0.0;
   Schlamm_Besch_Niv.Values[12] := 0.0;
   Schlamm_Besch_Niv.Values[13] := 0.0;
   Schlamm_Besch_Niv.Values[14] := 0.0;
   Schlamm_Besch_Niv.Values[15] := 0.0;
   Schlamm_Besch_Niv.Values[16] := 0.0;
   Schlamm_Besch_Niv.Values[17] := 0.0;
   Schlamm_Besch_Niv.Values[18] := 0.0;
   Schlamm_Besch_Niv.Values[19] := 0.0;
   Schlamm_Besch_Niv.Values[20] := 0.0;
   Schlamm_Besch_Niv.Values[21] := 0.0;
   Schlamm_Besch_Niv.Values[22] := 0.0;
   Schlamm_Besch_Niv.Values[23] := 0.0;
   Schlamm_Besch_Niv.Values[24] := 0.0;
   Schlamm_Besch_Niv.Values[25] := 0.0;
   Schlamm_Besch_Niv.Values[26] := 0.0;
   Schlamm_Besch_Niv.Values[27] := 0.0;
   Schlamm_Besch_Niv.Values[28] := 0.0;
   Schlamm_Besch_Niv.Values[29] := 0.0;
   Schlamm_Besch_Niv.Values[30] := 0.0;
   Schlamm_Besch_Niv.Values[31] := 0.0;
   Schlamm_Besch_Niv.Values[32] := 0.0;
   Schlamm_Besch_Niv.Values[33] := 0.0;
   Schlamm_Besch_Niv.Values[34] := 0.0;
   Schlamm_Besch_Niv.Values[35] := 0.0;
   Schlamm_Besch_Niv.Values[36] := 0.0;
   Schlamm_Besch_Niv.Values[37] := 0.0;
   Schlamm_Besch_Niv.Values[38] := 0.0;
   Schlamm_Besch_Niv.Values[39] := 0.0;
   Schlamm_Besch_Niv.Values[40] := 0.0;
   Schlamm_Besch_Niv.Values[41] := 0.0;
   Schlamm_Besch_Niv.Values[42] := 0.0;
   Schlamm_Besch_Niv.Values[43] := 0.0;
   Schlamm_Besch_Niv.Values[44] := 0.0;
   Schlamm_Besch_Niv.Values[45] := 0.0;
   Schlamm_Besch_Niv.Values[46] := 0.0;
   Schlamm_Besch_Niv.Values[47] := 0.0;
   Schlamm_Besch_Niv.Values[48] := 0.0;
   Schlamm_Besch_Niv.Values[49] := 0.0;
   Schlamm_Besch_Niv.Values[50] := 0.0;
   Schlamm_Besch_Niv.Values[51] := 0.0;
   Schlamm_Besch_Niv.Values[52] := 0.0;
   Schlamm_Besch_Niv.Values[53] := 0.0;
   Schlamm_Besch_Niv.Values[54] := 0.0;
   Schlamm_Besch_Niv.Values[55] := 0.0;
   Schlamm_Besch_Niv.Values[56] := 0.0;
   Schlamm_Besch_Niv.Values[57] := 0.0;
   Schlamm_Besch_Niv.Values[58] := 0.0;
   Schlamm_Besch_Niv.Values[59] := 0.0;
   Schlamm_Besch_Niv.Values[60] := 0.0;
   Schlamm_Besch_Niv.Values[61] := 0.0;
   Schlamm_Besch_Niv.Values[62] := 0.0;
   Schlamm_Besch_Niv.Values[63] := 0.0;
   Schlamm_Besch_Niv.Values[64] := 0.0;
   Schlamm_Besch_Niv.Values[65] := 0.0;
   Schlamm_Besch_Niv.Values[66] := 0.0;
   Schlamm_Besch_Niv.Values[67] := 0.0;
   Schlamm_Besch_Niv.Values[68] := 0.0;
   Schlamm_Besch_Niv.Values[69] := 0.0;
   Schlamm_Besch_Niv.Values[70] := 0.0;
   Schlamm_Besch_Niv.Values[71] := 0.0;
   Schlamm_Besch_Niv.Values[72] := 0.0;
   Schlamm_Besch_Niv.Values[73] := 0.0;
   Schlamm_Besch_Niv.Values[74] := 0.0;
   Schlamm_Besch_Niv.Values[75] := 0.0;
   Schlamm_Besch_Niv.Values[76] := 0.0;
   Schlamm_Besch_Niv.Values[77] := 0.0;
   Schlamm_Besch_Niv.Values[78] := 0.0;
   Schlamm_Besch_Niv.Values[79] := 0.0;
   Schlamm_Besch_Niv.Values[80] := 0.0;
   Schlamm_Besch_Niv.Values[81] := 0.0;
   Schlamm_Besch_Niv.Values[82] := 0.0;
   Schlamm_Besch_Niv.Values[83] := 0.0;
   Schlamm_Besch_Niv.Values[84] := 0.0;
   Schlamm_Besch_Niv.Values[85] := 0.0;
   Schlamm_Besch_Niv.Values[86] := 0.0;
   Schlamm_Besch_Niv.Values[87] := 0.0;
   Schlamm_Besch_Niv.Values[88] := 0.0;
   Schlamm_Besch_Niv.Values[89] := 0.0;
   Schlamm_Besch_Niv.Values[90] := 0.0;
   Schlamm_Besch_Niv.Values[91] := 0.0;
   Schlamm_Besch_Niv.Values[92] := 0.0;
   Schlamm_Besch_Niv.Values[93] := 0.0;
   Schlamm_Besch_Niv.Values[94] := 0.0;
   Schlamm_Besch_Niv.Values[95] := 0.0;
   Schlamm_Besch_Niv.Values[96] := 0.0;
   Schlamm_Besch_Niv.Values[97] := 0.0;
   Schlamm_Besch_Niv.Values[98] := 0.0;
   Schlamm_Besch_Niv.Values[99] := 0.0;
   Schlamm_Besch_Niv.Values[100] := 0.0;
   Schlamm_Besch_Niv.Values[101] := 0.0;
   Schlamm_Besch_Niv.Values[102] := 0.0;
   Schlamm_Besch_Niv.Values[103] := 0.0;
   Schlamm_Besch_Niv.Values[104] := 0.0;
   Schlamm_Besch_Niv.Values[105] := 0.0;
   Schlamm_Besch_Niv.Values[106] := 0.0;
   Schlamm_Besch_Niv.Values[107] := 0.0;
   Schlamm_Besch_Niv.Values[108] := 0.0;
   Schlamm_Besch_Niv.Values[109] := 0.0;
   Schlamm_Besch_Niv.Values[110] := 0.0;
   Schlamm_Besch_Niv.Values[111] := 0.0;
   Schlamm_Besch_Niv.Values[112] := 0.0;
   Schlamm_Besch_Niv.Values[113] := 0.0;
   Schlamm_Besch_Niv.Values[114] := 0.0;
   Schlamm_Besch_Niv.Values[115] := 0.0;
   Schlamm_Besch_Niv.Values[116] := 0.0;
   Schlamm_Besch_Niv.Values[117] := 0.0;
   Schlamm_Besch_Niv.Values[118] := 0.0;
   Schlamm_Besch_Niv.Values[119] := 0.0;
   Schlamm_Besch_DF.Values[0] := 0.0018084;
   Schlamm_Besch_DF.Values[1] := 0.0018084;
   Schlamm_Besch_DF.Values[2] := 0.0018084;
   Schlamm_Besch_DF.Values[3] := 0.0018084;
   Schlamm_Besch_DF.Values[4] := 0.0018084;
   Schlamm_Besch_DF.Values[5] := 0.0018084;
   Schlamm_Besch_DF.Values[6] := 0.0018084;
   Schlamm_Besch_DF.Values[7] := 0.0;
   Schlamm_Besch_DF.Values[8] := 0.0027126;
   Schlamm_Besch_DF.Values[9] := 0.0018084;
   Schlamm_Besch_DF.Values[10] := 0.0;
   Schlamm_Besch_DF.Values[11] := 0.0;
   Schlamm_Besch_DF.Values[12] := 0.0;
   Schlamm_Besch_DF.Values[13] := 0.0;
   Schlamm_Besch_DF.Values[14] := 0.0;
   Schlamm_Besch_DF.Values[15] := 0.0;
   Schlamm_Besch_DF.Values[16] := 0.0;
   Schlamm_Besch_DF.Values[17] := 0.0;
   Schlamm_Besch_DF.Values[18] := 0.0;
   Schlamm_Besch_DF.Values[19] := 0.0;
   Schlamm_Besch_DF.Values[20] := 0.0;
   Schlamm_Besch_DF.Values[21] := 0.0;
   Schlamm_Besch_DF.Values[22] := 0.0;
   Schlamm_Besch_DF.Values[23] := 0.0;
   Schlamm_Besch_DF.Values[24] := 0.0;
   Schlamm_Besch_DF.Values[25] := 0.0;
   Schlamm_Besch_DF.Values[26] := 0.0;
   Schlamm_Besch_DF.Values[27] := 0.0;
   Schlamm_Besch_DF.Values[28] := 0.0;
   Schlamm_Besch_DF.Values[29] := 0.0;
   Schlamm_Besch_DF.Values[30] := 0.0;
   Schlamm_Besch_DF.Values[31] := 0.0;
   Schlamm_Besch_DF.Values[32] := 0.0;
   Schlamm_Besch_DF.Values[33] := 0.0;
   Schlamm_Besch_DF.Values[34] := 0.0;
   Schlamm_Besch_DF.Values[35] := 0.0;
   Schlamm_Besch_DF.Values[36] := 0.0;
   Schlamm_Besch_DF.Values[37] := 0.0;
   Schlamm_Besch_DF.Values[38] := 0.0;
   Schlamm_Besch_DF.Values[39] := 0.0;
   Schlamm_Besch_DF.Values[40] := 0.0;
   Schlamm_Besch_DF.Values[41] := 0.0;
   Schlamm_Besch_DF.Values[42] := 0.0;
   Schlamm_Besch_DF.Values[43] := 0.0;
   Schlamm_Besch_DF.Values[44] := 0.0;
   Schlamm_Besch_DF.Values[45] := 0.0;
   Schlamm_Besch_DF.Values[46] := 0.0;
   Schlamm_Besch_DF.Values[47] := 0.0;
   Schlamm_Besch_DF.Values[48] := 0.0;
   Schlamm_Besch_DF.Values[49] := 0.0;
   Schlamm_Besch_DF.Values[50] := 0.0;
   Schlamm_Besch_DF.Values[51] := 0.0;
   Schlamm_Besch_DF.Values[52] := 0.0;
   Schlamm_Besch_DF.Values[53] := 0.0;
   Schlamm_Besch_DF.Values[54] := 0.0;
   Schlamm_Besch_DF.Values[55] := 0.0;
   Schlamm_Besch_DF.Values[56] := 0.0;
   Schlamm_Besch_DF.Values[57] := 0.0;
   Schlamm_Besch_DF.Values[58] := 0.0;
   Schlamm_Besch_DF.Values[59] := 0.0;
   Schlamm_Besch_DF.Values[60] := 0.0;
   Schlamm_Besch_DF.Values[61] := 0.0;
   Schlamm_Besch_DF.Values[62] := 0.0;
   Schlamm_Besch_DF.Values[63] := 0.0;
   Schlamm_Besch_DF.Values[64] := 0.0;
   Schlamm_Besch_DF.Values[65] := 0.0;
   Schlamm_Besch_DF.Values[66] := 0.0;
   Schlamm_Besch_DF.Values[67] := 0.0;
   Schlamm_Besch_DF.Values[68] := 0.0;
   Schlamm_Besch_DF.Values[69] := 0.0;
   Schlamm_Besch_DF.Values[70] := 0.0;
   Schlamm_Besch_DF.Values[71] := 0.0;
   Schlamm_Besch_DF.Values[72] := 0.0;
   Schlamm_Besch_DF.Values[73] := 0.0;
   Schlamm_Besch_DF.Values[74] := 0.0;
   Schlamm_Besch_DF.Values[75] := 0.0;
   Schlamm_Besch_DF.Values[76] := 0.0;
   Schlamm_Besch_DF.Values[77] := 0.0;
   Schlamm_Besch_DF.Values[78] := 0.0;
   Schlamm_Besch_DF.Values[79] := 0.0;
   Schlamm_Besch_DF.Values[80] := 0.0;
   Schlamm_Besch_DF.Values[81] := 0.0;
   Schlamm_Besch_DF.Values[82] := 0.0;
   Schlamm_Besch_DF.Values[83] := 0.0;
   Schlamm_Besch_DF.Values[84] := 0.0;
   Schlamm_Besch_DF.Values[85] := 0.0;
   Schlamm_Besch_DF.Values[86] := 0.0;
   Schlamm_Besch_DF.Values[87] := 0.0;
   Schlamm_Besch_DF.Values[88] := 0.0;
   Schlamm_Besch_DF.Values[89] := 0.0;
   Schlamm_Besch_DF.Values[90] := 0.0;
   Schlamm_Besch_DF.Values[91] := 0.0;
   Schlamm_Besch_DF.Values[92] := 0.0;
   Schlamm_Besch_DF.Values[93] := 0.0;
   Schlamm_Besch_DF.Values[94] := 0.0;
   Schlamm_Besch_DF.Values[95] := 0.0;
   Schlamm_Besch_DF.Values[96] := 0.0;
   Schlamm_Besch_DF.Values[97] := 0.0;
   Schlamm_Besch_DF.Values[98] := 0.0;
   Schlamm_Besch_DF.Values[99] := 0.0;
   Schlamm_Besch_DF.Values[100] := 0.0;
   Schlamm_Besch_DF.Values[101] := 0.0;
   Schlamm_Besch_DF.Values[102] := 0.0;
   Schlamm_Besch_DF.Values[103] := 0.0;
   Schlamm_Besch_DF.Values[104] := 0.0;
   Schlamm_Besch_DF.Values[105] := 0.0;
   Schlamm_Besch_DF.Values[106] := 0.0;
   Schlamm_Besch_DF.Values[107] := 0.0;
   Schlamm_Besch_DF.Values[108] := 0.0;
   Schlamm_Besch_DF.Values[109] := 0.0;
   Schlamm_Besch_DF.Values[110] := 0.0;
   Schlamm_Besch_DF.Values[111] := 0.0;
   Schlamm_Besch_DF.Values[112] := 0.0;
   Schlamm_Besch_DF.Values[113] := 0.0;
   Schlamm_Besch_DF.Values[114] := 0.0;
   Schlamm_Besch_DF.Values[115] := 0.0;
   Schlamm_Besch_DF.Values[116] := 0.0;
   Schlamm_Besch_DF.Values[117] := 0.0;
   Schlamm_Besch_DF.Values[118] := 0.0;
   Schlamm_Besch_DF.Values[119] := 0.0;
   Truebwasser_Niv.Values[0] := 26.07261;
   Truebwasser_Niv.Values[1] := 26.07713;
   Truebwasser_Niv.Values[2] := 26.07713;
   Truebwasser_Niv.Values[3] := 26.07713;
   Truebwasser_Niv.Values[4] := 26.07713;
   Truebwasser_Niv.Values[5] := 26.14494;
   Truebwasser_Niv.Values[6] := 26.14946;
   Truebwasser_Niv.Values[7] := 26.07261;
   Truebwasser_Niv.Values[8] := 26.07261;
   Truebwasser_Niv.Values[9] := 26.07261;
   Truebwasser_Niv.Values[10] := 0.0;
   Truebwasser_Niv.Values[11] := 0.0;
   Truebwasser_Niv.Values[12] := 0.0;
   Truebwasser_Niv.Values[13] := 0.0;
   Truebwasser_Niv.Values[14] := 0.0;
   Truebwasser_Niv.Values[15] := 0.0;
   Truebwasser_Niv.Values[16] := 0.0;
   Truebwasser_Niv.Values[17] := 0.0;
   Truebwasser_Niv.Values[18] := 0.0;
   Truebwasser_Niv.Values[19] := 0.0;
   Truebwasser_Niv.Values[20] := 0.0;
   Truebwasser_Niv.Values[21] := 0.0;
   Truebwasser_Niv.Values[22] := 0.0;
   Truebwasser_Niv.Values[23] := 0.0;
   Truebwasser_Niv.Values[24] := 0.0;
   Truebwasser_Niv.Values[25] := 0.0;
   Truebwasser_Niv.Values[26] := 0.0;
   Truebwasser_Niv.Values[27] := 0.0;
   Truebwasser_Niv.Values[28] := 0.0;
   Truebwasser_Niv.Values[29] := 0.0;
   Truebwasser_Niv.Values[30] := 0.0;
   Truebwasser_Niv.Values[31] := 0.0;
   Truebwasser_Niv.Values[32] := 0.0;
   Truebwasser_Niv.Values[33] := 0.0;
   Truebwasser_Niv.Values[34] := 0.0;
   Truebwasser_Niv.Values[35] := 0.0;
   Truebwasser_Niv.Values[36] := 0.0;
   Truebwasser_Niv.Values[37] := 0.0;
   Truebwasser_Niv.Values[38] := 0.0;
   Truebwasser_Niv.Values[39] := 0.0;
   Truebwasser_Niv.Values[40] := 0.0;
   Truebwasser_Niv.Values[41] := 0.0;
   Truebwasser_Niv.Values[42] := 0.0;
   Truebwasser_Niv.Values[43] := 0.0;
   Truebwasser_Niv.Values[44] := 0.0;
   Truebwasser_Niv.Values[45] := 0.0;
   Truebwasser_Niv.Values[46] := 0.0;
   Truebwasser_Niv.Values[47] := 0.0;
   Truebwasser_Niv.Values[48] := 0.0;
   Truebwasser_Niv.Values[49] := 0.0;
   Truebwasser_Niv.Values[50] := 0.0;
   Truebwasser_Niv.Values[51] := 0.0;
   Truebwasser_Niv.Values[52] := 0.0;
   Truebwasser_Niv.Values[53] := 0.0;
   Truebwasser_Niv.Values[54] := 0.0;
   Truebwasser_Niv.Values[55] := 0.0;
   Truebwasser_Niv.Values[56] := 0.0;
   Truebwasser_Niv.Values[57] := 0.0;
   Truebwasser_Niv.Values[58] := 0.0;
   Truebwasser_Niv.Values[59] := 0.0;
   Truebwasser_Niv.Values[60] := 0.0;
   Truebwasser_Niv.Values[61] := 0.0;
   Truebwasser_Niv.Values[62] := 0.0;
   Truebwasser_Niv.Values[63] := 0.0;
   Truebwasser_Niv.Values[64] := 0.0;
   Truebwasser_Niv.Values[65] := 0.0;
   Truebwasser_Niv.Values[66] := 0.0;
   Truebwasser_Niv.Values[67] := 0.0;
   Truebwasser_Niv.Values[68] := 0.0;
   Truebwasser_Niv.Values[69] := 0.0;
   Truebwasser_Niv.Values[70] := 0.0;
   Truebwasser_Niv.Values[71] := 0.0;
   Truebwasser_Niv.Values[72] := 0.0;
   Truebwasser_Niv.Values[73] := 0.0;
   Truebwasser_Niv.Values[74] := 0.0;
   Truebwasser_Niv.Values[75] := 0.0;
   Truebwasser_Niv.Values[76] := 0.0;
   Truebwasser_Niv.Values[77] := 0.0;
   Truebwasser_Niv.Values[78] := 0.0;
   Truebwasser_Niv.Values[79] := 0.0;
   Truebwasser_Niv.Values[80] := 0.0;
   Truebwasser_Niv.Values[81] := 0.0;
   Truebwasser_Niv.Values[82] := 0.0;
   Truebwasser_Niv.Values[83] := 0.0;
   Truebwasser_Niv.Values[84] := 0.0;
   Truebwasser_Niv.Values[85] := 0.0;
   Truebwasser_Niv.Values[86] := 0.0;
   Truebwasser_Niv.Values[87] := 0.0;
   Truebwasser_Niv.Values[88] := 0.0;
   Truebwasser_Niv.Values[89] := 0.0;
   Truebwasser_Niv.Values[90] := 0.0;
   Truebwasser_Niv.Values[91] := 0.0;
   Truebwasser_Niv.Values[92] := 0.0;
   Truebwasser_Niv.Values[93] := 0.0;
   Truebwasser_Niv.Values[94] := 0.0;
   Truebwasser_Niv.Values[95] := 0.0;
   Truebwasser_Niv.Values[96] := 0.0;
   Truebwasser_Niv.Values[97] := 0.0;
   Truebwasser_Niv.Values[98] := 0.0;
   Truebwasser_Niv.Values[99] := 0.0;
   Truebwasser_Niv.Values[100] := 0.0;
   Truebwasser_Niv.Values[101] := 0.0;
   Truebwasser_Niv.Values[102] := 0.0;
   Truebwasser_Niv.Values[103] := 0.0;
   Truebwasser_Niv.Values[104] := 0.0;
   Truebwasser_Niv.Values[105] := 0.0;
   Truebwasser_Niv.Values[106] := 0.0;
   Truebwasser_Niv.Values[107] := 0.0;
   Truebwasser_Niv.Values[108] := 0.0;
   Truebwasser_Niv.Values[109] := 0.0;
   Truebwasser_Niv.Values[110] := 0.0;
   Truebwasser_Niv.Values[111] := 0.0;
   Truebwasser_Niv.Values[112] := 0.0;
   Truebwasser_Niv.Values[113] := 0.0;
   Truebwasser_Niv.Values[114] := 0.0;
   Truebwasser_Niv.Values[115] := 0.0;
   Truebwasser_Niv.Values[116] := 0.0;
   Truebwasser_Niv.Values[117] := 0.0;
   Truebwasser_Niv.Values[118] := 0.0;
   Truebwasser_Niv.Values[119] := 0.0;
   Truebwasser_DF.Values[0] := -0.0022605;
   Truebwasser_DF.Values[1] := -0.0022605;
   Truebwasser_DF.Values[2] := -0.0022605;
   Truebwasser_DF.Values[3] := -0.0022605;
   Truebwasser_DF.Values[4] := -0.0022605;
   Truebwasser_DF.Values[5] := -0.0022605;
   Truebwasser_DF.Values[6] := -0.0022605;
   Truebwasser_DF.Values[7] := -0.0022605;
   Truebwasser_DF.Values[8] := -0.0022605;
   Truebwasser_DF.Values[9] := -0.0022605;
   Truebwasser_DF.Values[10] := 0.0;
   Truebwasser_DF.Values[11] := 0.0;
   Truebwasser_DF.Values[12] := 0.0;
   Truebwasser_DF.Values[13] := 0.0;
   Truebwasser_DF.Values[14] := 0.0;
   Truebwasser_DF.Values[15] := 0.0;
   Truebwasser_DF.Values[16] := 0.0;
   Truebwasser_DF.Values[17] := 0.0;
   Truebwasser_DF.Values[18] := 0.0;
   Truebwasser_DF.Values[19] := 0.0;
   Truebwasser_DF.Values[20] := 0.0;
   Truebwasser_DF.Values[21] := 0.0;
   Truebwasser_DF.Values[22] := 0.0;
   Truebwasser_DF.Values[23] := 0.0;
   Truebwasser_DF.Values[24] := 0.0;
   Truebwasser_DF.Values[25] := 0.0;
   Truebwasser_DF.Values[26] := 0.0;
   Truebwasser_DF.Values[27] := 0.0;
   Truebwasser_DF.Values[28] := 0.0;
   Truebwasser_DF.Values[29] := 0.0;
   Truebwasser_DF.Values[30] := 0.0;
   Truebwasser_DF.Values[31] := 0.0;
   Truebwasser_DF.Values[32] := 0.0;
   Truebwasser_DF.Values[33] := 0.0;
   Truebwasser_DF.Values[34] := 0.0;
   Truebwasser_DF.Values[35] := 0.0;
   Truebwasser_DF.Values[36] := 0.0;
   Truebwasser_DF.Values[37] := 0.0;
   Truebwasser_DF.Values[38] := 0.0;
   Truebwasser_DF.Values[39] := 0.0;
   Truebwasser_DF.Values[40] := 0.0;
   Truebwasser_DF.Values[41] := 0.0;
   Truebwasser_DF.Values[42] := 0.0;
   Truebwasser_DF.Values[43] := 0.0;
   Truebwasser_DF.Values[44] := 0.0;
   Truebwasser_DF.Values[45] := 0.0;
   Truebwasser_DF.Values[46] := 0.0;
   Truebwasser_DF.Values[47] := 0.0;
   Truebwasser_DF.Values[48] := 0.0;
   Truebwasser_DF.Values[49] := 0.0;
   Truebwasser_DF.Values[50] := 0.0;
   Truebwasser_DF.Values[51] := 0.0;
   Truebwasser_DF.Values[52] := 0.0;
   Truebwasser_DF.Values[53] := 0.0;
   Truebwasser_DF.Values[54] := 0.0;
   Truebwasser_DF.Values[55] := 0.0;
   Truebwasser_DF.Values[56] := 0.0;
   Truebwasser_DF.Values[57] := 0.0;
   Truebwasser_DF.Values[58] := 0.0;
   Truebwasser_DF.Values[59] := 0.0;
   Truebwasser_DF.Values[60] := 0.0;
   Truebwasser_DF.Values[61] := 0.0;
   Truebwasser_DF.Values[62] := 0.0;
   Truebwasser_DF.Values[63] := 0.0;
   Truebwasser_DF.Values[64] := 0.0;
   Truebwasser_DF.Values[65] := 0.0;
   Truebwasser_DF.Values[66] := 0.0;
   Truebwasser_DF.Values[67] := 0.0;
   Truebwasser_DF.Values[68] := 0.0;
   Truebwasser_DF.Values[69] := 0.0;
   Truebwasser_DF.Values[70] := 0.0;
   Truebwasser_DF.Values[71] := 0.0;
   Truebwasser_DF.Values[72] := 0.0;
   Truebwasser_DF.Values[73] := 0.0;
   Truebwasser_DF.Values[74] := 0.0;
   Truebwasser_DF.Values[75] := 0.0;
   Truebwasser_DF.Values[76] := 0.0;
   Truebwasser_DF.Values[77] := 0.0;
   Truebwasser_DF.Values[78] := 0.0;
   Truebwasser_DF.Values[79] := 0.0;
   Truebwasser_DF.Values[80] := 0.0;
   Truebwasser_DF.Values[81] := 0.0;
   Truebwasser_DF.Values[82] := 0.0;
   Truebwasser_DF.Values[83] := 0.0;
   Truebwasser_DF.Values[84] := 0.0;
   Truebwasser_DF.Values[85] := 0.0;
   Truebwasser_DF.Values[86] := 0.0;
   Truebwasser_DF.Values[87] := 0.0;
   Truebwasser_DF.Values[88] := 0.0;
   Truebwasser_DF.Values[89] := 0.0;
   Truebwasser_DF.Values[90] := 0.0;
   Truebwasser_DF.Values[91] := 0.0;
   Truebwasser_DF.Values[92] := 0.0;
   Truebwasser_DF.Values[93] := 0.0;
   Truebwasser_DF.Values[94] := 0.0;
   Truebwasser_DF.Values[95] := 0.0;
   Truebwasser_DF.Values[96] := 0.0;
   Truebwasser_DF.Values[97] := 0.0;
   Truebwasser_DF.Values[98] := 0.0;
   Truebwasser_DF.Values[99] := 0.0;
   Truebwasser_DF.Values[100] := 0.0;
   Truebwasser_DF.Values[101] := 0.0;
   Truebwasser_DF.Values[102] := 0.0;
   Truebwasser_DF.Values[103] := 0.0;
   Truebwasser_DF.Values[104] := 0.0;
   Truebwasser_DF.Values[105] := 0.0;
   Truebwasser_DF.Values[106] := 0.0;
   Truebwasser_DF.Values[107] := 0.0;
   Truebwasser_DF.Values[108] := 0.0;
   Truebwasser_DF.Values[109] := 0.0;
   Truebwasser_DF.Values[110] := 0.0;
   Truebwasser_DF.Values[111] := 0.0;
   Truebwasser_DF.Values[112] := 0.0;
   Truebwasser_DF.Values[113] := 0.0;
   Truebwasser_DF.Values[114] := 0.0;
   Truebwasser_DF.Values[115] := 0.0;
   Truebwasser_DF.Values[116] := 0.0;
   Truebwasser_DF.Values[117] := 0.0;
   Truebwasser_DF.Values[118] := 0.0;
   Truebwasser_DF.Values[119] := 0.0;
   Zulauf_SF_Niv.Values[0] := 0.0;
   Zulauf_SF_Niv.Values[1] := 0.0;
   Zulauf_SF_Niv.Values[2] := 0.0;
   Zulauf_SF_Niv.Values[3] := 0.0;
   Zulauf_SF_Niv.Values[4] := 0.0;
   Zulauf_SF_Niv.Values[5] := 0.0;
   Zulauf_SF_Niv.Values[6] := 0.0;
   Zulauf_SF_Niv.Values[7] := 0.0;
   Zulauf_SF_Niv.Values[8] := 0.0;
   Zulauf_SF_Niv.Values[9] := 0.0;
   Zulauf_SF_Niv.Values[10] := 0.0;
   Zulauf_SF_Niv.Values[11] := 0.0;
   Zulauf_SF_Niv.Values[12] := 0.0;
   Zulauf_SF_Niv.Values[13] := 0.0;
   Zulauf_SF_Niv.Values[14] := 0.0;
   Zulauf_SF_Niv.Values[15] := 0.0;
   Zulauf_SF_Niv.Values[16] := 0.0;
   Zulauf_SF_Niv.Values[17] := 0.0;
   Zulauf_SF_Niv.Values[18] := 0.0;
   Zulauf_SF_Niv.Values[19] := 0.0;
   Zulauf_SF_Niv.Values[20] := 0.0;
   Zulauf_SF_Niv.Values[21] := 0.0;
   Zulauf_SF_Niv.Values[22] := 0.0;
   Zulauf_SF_Niv.Values[23] := 0.0;
   Zulauf_SF_Niv.Values[24] := 0.0;
   Zulauf_SF_Niv.Values[25] := 0.0;
   Zulauf_SF_Niv.Values[26] := 0.0;
   Zulauf_SF_Niv.Values[27] := 0.0;
   Zulauf_SF_Niv.Values[28] := 0.0;
   Zulauf_SF_Niv.Values[29] := 0.0;
   Zulauf_SF_Niv.Values[30] := 0.0;
   Zulauf_SF_Niv.Values[31] := 0.0;
   Zulauf_SF_Niv.Values[32] := 0.0;
   Zulauf_SF_Niv.Values[33] := 0.0;
   Zulauf_SF_Niv.Values[34] := 0.0;
   Zulauf_SF_Niv.Values[35] := 0.0;
   Zulauf_SF_Niv.Values[36] := 0.0;
   Zulauf_SF_Niv.Values[37] := 0.0;
   Zulauf_SF_Niv.Values[38] := 0.0;
   Zulauf_SF_Niv.Values[39] := 0.0;
   Zulauf_SF_Niv.Values[40] := 0.0;
   Zulauf_SF_Niv.Values[41] := 0.0;
   Zulauf_SF_Niv.Values[42] := 0.0;
   Zulauf_SF_Niv.Values[43] := 0.0;
   Zulauf_SF_Niv.Values[44] := 0.0;
   Zulauf_SF_Niv.Values[45] := 0.0;
   Zulauf_SF_Niv.Values[46] := 0.0;
   Zulauf_SF_Niv.Values[47] := 0.0;
   Zulauf_SF_Niv.Values[48] := 0.0;
   Zulauf_SF_Niv.Values[49] := 0.0;
   Zulauf_SF_Niv.Values[50] := 0.0;
   Zulauf_SF_Niv.Values[51] := 0.0;
   Zulauf_SF_Niv.Values[52] := 0.0;
   Zulauf_SF_Niv.Values[53] := 0.0;
   Zulauf_SF_Niv.Values[54] := 0.0;
   Zulauf_SF_Niv.Values[55] := 0.0;
   Zulauf_SF_Niv.Values[56] := 0.0;
   Zulauf_SF_Niv.Values[57] := 0.0;
   Zulauf_SF_Niv.Values[58] := 0.0;
   Zulauf_SF_Niv.Values[59] := 0.0;
   Zulauf_SF_Niv.Values[60] := 0.0;
   Zulauf_SF_Niv.Values[61] := 0.0;
   Zulauf_SF_Niv.Values[62] := 0.0;
   Zulauf_SF_Niv.Values[63] := 0.0;
   Zulauf_SF_Niv.Values[64] := 0.0;
   Zulauf_SF_Niv.Values[65] := 0.0;
   Zulauf_SF_Niv.Values[66] := 0.0;
   Zulauf_SF_Niv.Values[67] := 0.0;
   Zulauf_SF_Niv.Values[68] := 0.0;
   Zulauf_SF_Niv.Values[69] := 0.0;
   Zulauf_SF_Niv.Values[70] := 0.0;
   Zulauf_SF_Niv.Values[71] := 0.0;
   Zulauf_SF_Niv.Values[72] := 0.0;
   Zulauf_SF_Niv.Values[73] := 0.0;
   Zulauf_SF_Niv.Values[74] := 0.0;
   Zulauf_SF_Niv.Values[75] := 0.0;
   Zulauf_SF_Niv.Values[76] := 0.0;
   Zulauf_SF_Niv.Values[77] := 0.0;
   Zulauf_SF_Niv.Values[78] := 0.0;
   Zulauf_SF_Niv.Values[79] := 0.0;
   Zulauf_SF_Niv.Values[80] := 0.0;
   Zulauf_SF_Niv.Values[81] := 0.0;
   Zulauf_SF_Niv.Values[82] := 0.0;
   Zulauf_SF_Niv.Values[83] := 0.0;
   Zulauf_SF_Niv.Values[84] := 0.0;
   Zulauf_SF_Niv.Values[85] := 0.0;
   Zulauf_SF_Niv.Values[86] := 0.0;
   Zulauf_SF_Niv.Values[87] := 0.0;
   Zulauf_SF_Niv.Values[88] := 0.0;
   Zulauf_SF_Niv.Values[89] := 0.0;
   Zulauf_SF_Niv.Values[90] := 0.0;
   Zulauf_SF_Niv.Values[91] := 0.0;
   Zulauf_SF_Niv.Values[92] := 0.0;
   Zulauf_SF_Niv.Values[93] := 0.0;
   Zulauf_SF_Niv.Values[94] := 0.0;
   Zulauf_SF_Niv.Values[95] := 0.0;
   Zulauf_SF_Niv.Values[96] := 0.0;
   Zulauf_SF_Niv.Values[97] := 0.0;
   Zulauf_SF_Niv.Values[98] := 0.0;
   Zulauf_SF_Niv.Values[99] := 0.0;
   Zulauf_SF_Niv.Values[100] := 0.0;
   Zulauf_SF_Niv.Values[101] := 0.0;
   Zulauf_SF_Niv.Values[102] := 0.0;
   Zulauf_SF_Niv.Values[103] := 0.0;
   Zulauf_SF_Niv.Values[104] := 0.0;
   Zulauf_SF_Niv.Values[105] := 0.0;
   Zulauf_SF_Niv.Values[106] := 0.0;
   Zulauf_SF_Niv.Values[107] := 0.0;
   Zulauf_SF_Niv.Values[108] := 0.0;
   Zulauf_SF_Niv.Values[109] := 0.0;
   Zulauf_SF_Niv.Values[110] := 0.0;
   Zulauf_SF_Niv.Values[111] := 0.0;
   Zulauf_SF_Niv.Values[112] := 0.0;
   Zulauf_SF_Niv.Values[113] := 0.0;
   Zulauf_SF_Niv.Values[114] := 0.0;
   Zulauf_SF_Niv.Values[115] := 0.0;
   Zulauf_SF_Niv.Values[116] := 0.0;
   Zulauf_SF_Niv.Values[117] := 0.0;
   Zulauf_SF_Niv.Values[118] := 0.0;
   Zulauf_SF_Niv.Values[119] := 0.0;
   Ablauf_NOx.Values[0] := 1.462996;
   Ablauf_NOx.Values[1] := 1.462996;
   Ablauf_NOx.Values[2] := 1.462996;
   Ablauf_NOx.Values[3] := 1.462996;
   Ablauf_NOx.Values[4] := 1.462996;
   Ablauf_NOx.Values[5] := 1.462996;
   Ablauf_NOx.Values[6] := 1.462996;
   Ablauf_NOx.Values[7] := 1.462996;
   Ablauf_NOx.Values[8] := 1.462996;
   Ablauf_NOx.Values[9] := 1.462996;
   Ablauf_NOx.Values[10] := 1.462996;
   Ablauf_NOx.Values[11] := 1.462996;
   Ablauf_NOx.Values[12] := 1.462996;
   Ablauf_NOx.Values[13] := 1.462996;
   Ablauf_NOx.Values[14] := 1.462996;
   Ablauf_NOx.Values[15] := 1.462996;
   Ablauf_NOx.Values[16] := 1.462996;
   Ablauf_NOx.Values[17] := 1.462996;
   Ablauf_NOx.Values[18] := 1.462996;
   Ablauf_NOx.Values[19] := 1.462996;
   Ablauf_NOx.Values[20] := 1.462996;
   Ablauf_NOx.Values[21] := 1.462996;
   Ablauf_NOx.Values[22] := 1.462996;
   Ablauf_NOx.Values[23] := 1.462996;
   Ablauf_NOx.Values[24] := 1.462996;
   Ablauf_NOx.Values[25] := 1.462996;
   Ablauf_NOx.Values[26] := 1.462996;
   Ablauf_NOx.Values[27] := 1.462996;
   Ablauf_NOx.Values[28] := 1.462996;
   Ablauf_NOx.Values[29] := 1.462996;
   Ablauf_NOx.Values[30] := 0.0;
   Ablauf_NOx.Values[31] := 0.0;
   Ablauf_NOx.Values[32] := 0.0;
   Ablauf_NOx.Values[33] := 0.0;
   Ablauf_NOx.Values[34] := 0.0;
   Ablauf_NOx.Values[35] := 0.0;
   Ablauf_NOx.Values[36] := 0.0;
   Ablauf_NOx.Values[37] := 0.0;
   Ablauf_NOx.Values[38] := 0.0;
   Ablauf_NOx.Values[39] := 0.0;
   Ablauf_NOx.Values[40] := 0.0;
   Ablauf_NOx.Values[41] := 0.0;
   Ablauf_NOx.Values[42] := 0.0;
   Ablauf_NOx.Values[43] := 0.0;
   Ablauf_NOx.Values[44] := 0.0;
   Ablauf_NOx.Values[45] := 0.0;
   Ablauf_NOx.Values[46] := 0.0;
   Ablauf_NOx.Values[47] := 0.0;
   Ablauf_NOx.Values[48] := 0.0;
   Ablauf_NOx.Values[49] := 0.0;
   Ablauf_NOx.Values[50] := 0.0;
   Ablauf_NOx.Values[51] := 0.0;
   Ablauf_NOx.Values[52] := 0.0;
   Ablauf_NOx.Values[53] := 0.0;
   Ablauf_NOx.Values[54] := 0.0;
   Ablauf_NOx.Values[55] := 0.0;
   Ablauf_NOx.Values[56] := 0.0;
   Ablauf_NOx.Values[57] := 0.0;
   Ablauf_NOx.Values[58] := 0.0;
   Ablauf_NOx.Values[59] := 0.0;
   Ablauf_NOx.Values[60] := 0.0;
   Ablauf_NOx.Values[61] := 0.0;
   Ablauf_NOx.Values[62] := 0.0;
   Ablauf_NOx.Values[63] := 0.0;
   Ablauf_NOx.Values[64] := 0.0;
   Ablauf_NOx.Values[65] := 0.0;
   Ablauf_NOx.Values[66] := 0.0;
   Ablauf_NOx.Values[67] := 0.0;
   Ablauf_NOx.Values[68] := 0.0;
   Ablauf_NOx.Values[69] := 0.0;
   Ablauf_NOx.Values[70] := 0.0;
   Ablauf_NOx.Values[71] := 0.0;
   Ablauf_NOx.Values[72] := 0.0;
   Ablauf_NOx.Values[73] := 0.0;
   Ablauf_NOx.Values[74] := 0.0;
   Ablauf_NOx.Values[75] := 0.0;
   Ablauf_NOx.Values[76] := 0.0;
   Ablauf_NOx.Values[77] := 0.0;
   Ablauf_NOx.Values[78] := 0.0;
   Ablauf_NOx.Values[79] := 0.0;
   Ablauf_NOx.Values[80] := 0.0;
   Ablauf_NOx.Values[81] := 0.0;
   Ablauf_NOx.Values[82] := 0.0;
   Ablauf_NOx.Values[83] := 0.0;
   Ablauf_NOx.Values[84] := 0.0;
   Ablauf_NOx.Values[85] := 0.0;
   Ablauf_NOx.Values[86] := 0.0;
   Ablauf_NOx.Values[87] := 0.0;
   Ablauf_NOx.Values[88] := 0.0;
   Ablauf_NOx.Values[89] := 0.0;
   Ablauf_NOx.Values[90] := 0.0;
   Ablauf_NOx.Values[91] := 0.0;
   Ablauf_NOx.Values[92] := 0.0;
   Ablauf_NOx.Values[93] := 0.0;
   Ablauf_NOx.Values[94] := 0.0;
   Ablauf_NOx.Values[95] := 0.0;
   Ablauf_NOx.Values[96] := 0.0;
   Ablauf_NOx.Values[97] := 0.0;
   Ablauf_NOx.Values[98] := 0.0;
   Ablauf_NOx.Values[99] := 0.0;
   Ablauf_NOx.Values[100] := 0.0;
   Ablauf_NOx.Values[101] := 0.0;
   Ablauf_NOx.Values[102] := 0.0;
   Ablauf_NOx.Values[103] := 0.0;
   Ablauf_NOx.Values[104] := 0.0;
   Ablauf_NOx.Values[105] := 0.0;
   Ablauf_NOx.Values[106] := 0.0;
   Ablauf_NOx.Values[107] := 0.0;
   Ablauf_NOx.Values[108] := 0.0;
   Ablauf_NOx.Values[109] := 0.0;
   Ablauf_NOx.Values[110] := 0.0;
   Ablauf_NOx.Values[111] := 0.0;
   Ablauf_NOx.Values[112] := 0.0;
   Ablauf_NOx.Values[113] := 0.0;
   Ablauf_NOx.Values[114] := 0.0;
   Ablauf_NOx.Values[115] := 0.0;
   Ablauf_NOx.Values[116] := 0.0;
   Ablauf_NOx.Values[117] := 0.0;
   Ablauf_NOx.Values[118] := 0.0;
   Ablauf_NOx.Values[119] := 0.0;
   Ablauf_PO4.Values[0] := 2.762331;
   Ablauf_PO4.Values[1] := 2.762331;
   Ablauf_PO4.Values[2] := 2.762331;
   Ablauf_PO4.Values[3] := 2.762331;
   Ablauf_PO4.Values[4] := 2.762331;
   Ablauf_PO4.Values[5] := 2.762331;
   Ablauf_PO4.Values[6] := 2.762331;
   Ablauf_PO4.Values[7] := 2.762331;
   Ablauf_PO4.Values[8] := 2.762331;
   Ablauf_PO4.Values[9] := 2.762331;
   Ablauf_PO4.Values[10] := 2.762331;
   Ablauf_PO4.Values[11] := 2.762331;
   Ablauf_PO4.Values[12] := 2.762331;
   Ablauf_PO4.Values[13] := 2.762331;
   Ablauf_PO4.Values[14] := 2.762331;
   Ablauf_PO4.Values[15] := 2.762331;
   Ablauf_PO4.Values[16] := 2.762331;
   Ablauf_PO4.Values[17] := 2.762331;
   Ablauf_PO4.Values[18] := 2.762331;
   Ablauf_PO4.Values[19] := 2.762331;
   Ablauf_PO4.Values[20] := 2.762331;
   Ablauf_PO4.Values[21] := 2.762331;
   Ablauf_PO4.Values[22] := 2.762331;
   Ablauf_PO4.Values[23] := 2.762331;
   Ablauf_PO4.Values[24] := 2.762331;
   Ablauf_PO4.Values[25] := 2.762331;
   Ablauf_PO4.Values[26] := 2.762331;
   Ablauf_PO4.Values[27] := 2.762331;
   Ablauf_PO4.Values[28] := 2.762331;
   Ablauf_PO4.Values[29] := 2.762331;
   Ablauf_PO4.Values[30] := 0.0;
   Ablauf_PO4.Values[31] := 0.0;
   Ablauf_PO4.Values[32] := 0.0;
   Ablauf_PO4.Values[33] := 0.0;
   Ablauf_PO4.Values[34] := 0.0;
   Ablauf_PO4.Values[35] := 0.0;
   Ablauf_PO4.Values[36] := 0.0;
   Ablauf_PO4.Values[37] := 0.0;
   Ablauf_PO4.Values[38] := 0.0;
   Ablauf_PO4.Values[39] := 0.0;
   Ablauf_PO4.Values[40] := 0.0;
   Ablauf_PO4.Values[41] := 0.0;
   Ablauf_PO4.Values[42] := 0.0;
   Ablauf_PO4.Values[43] := 0.0;
   Ablauf_PO4.Values[44] := 0.0;
   Ablauf_PO4.Values[45] := 0.0;
   Ablauf_PO4.Values[46] := 0.0;
   Ablauf_PO4.Values[47] := 0.0;
   Ablauf_PO4.Values[48] := 0.0;
   Ablauf_PO4.Values[49] := 0.0;
   Ablauf_PO4.Values[50] := 0.0;
   Ablauf_PO4.Values[51] := 0.0;
   Ablauf_PO4.Values[52] := 0.0;
   Ablauf_PO4.Values[53] := 0.0;
   Ablauf_PO4.Values[54] := 0.0;
   Ablauf_PO4.Values[55] := 0.0;
   Ablauf_PO4.Values[56] := 0.0;
   Ablauf_PO4.Values[57] := 0.0;
   Ablauf_PO4.Values[58] := 0.0;
   Ablauf_PO4.Values[59] := 0.0;
   Ablauf_PO4.Values[60] := 0.0;
   Ablauf_PO4.Values[61] := 0.0;
   Ablauf_PO4.Values[62] := 0.0;
   Ablauf_PO4.Values[63] := 0.0;
   Ablauf_PO4.Values[64] := 0.0;
   Ablauf_PO4.Values[65] := 0.0;
   Ablauf_PO4.Values[66] := 0.0;
   Ablauf_PO4.Values[67] := 0.0;
   Ablauf_PO4.Values[68] := 0.0;
   Ablauf_PO4.Values[69] := 0.0;
   Ablauf_PO4.Values[70] := 0.0;
   Ablauf_PO4.Values[71] := 0.0;
   Ablauf_PO4.Values[72] := 0.0;
   Ablauf_PO4.Values[73] := 0.0;
   Ablauf_PO4.Values[74] := 0.0;
   Ablauf_PO4.Values[75] := 0.0;
   Ablauf_PO4.Values[76] := 0.0;
   Ablauf_PO4.Values[77] := 0.0;
   Ablauf_PO4.Values[78] := 0.0;
   Ablauf_PO4.Values[79] := 0.0;
   Ablauf_PO4.Values[80] := 0.0;
   Ablauf_PO4.Values[81] := 0.0;
   Ablauf_PO4.Values[82] := 0.0;
   Ablauf_PO4.Values[83] := 0.0;
   Ablauf_PO4.Values[84] := 0.0;
   Ablauf_PO4.Values[85] := 0.0;
   Ablauf_PO4.Values[86] := 0.0;
   Ablauf_PO4.Values[87] := 0.0;
   Ablauf_PO4.Values[88] := 0.0;
   Ablauf_PO4.Values[89] := 0.0;
   Ablauf_PO4.Values[90] := 0.0;
   Ablauf_PO4.Values[91] := 0.0;
   Ablauf_PO4.Values[92] := 0.0;
   Ablauf_PO4.Values[93] := 0.0;
   Ablauf_PO4.Values[94] := 0.0;
   Ablauf_PO4.Values[95] := 0.0;
   Ablauf_PO4.Values[96] := 0.0;
   Ablauf_PO4.Values[97] := 0.0;
   Ablauf_PO4.Values[98] := 0.0;
   Ablauf_PO4.Values[99] := 0.0;
   Ablauf_PO4.Values[100] := 0.0;
   Ablauf_PO4.Values[101] := 0.0;
   Ablauf_PO4.Values[102] := 0.0;
   Ablauf_PO4.Values[103] := 0.0;
   Ablauf_PO4.Values[104] := 0.0;
   Ablauf_PO4.Values[105] := 0.0;
   Ablauf_PO4.Values[106] := 0.0;
   Ablauf_PO4.Values[107] := 0.0;
   Ablauf_PO4.Values[108] := 0.0;
   Ablauf_PO4.Values[109] := 0.0;
   Ablauf_PO4.Values[110] := 0.0;
   Ablauf_PO4.Values[111] := 0.0;
   Ablauf_PO4.Values[112] := 0.0;
   Ablauf_PO4.Values[113] := 0.0;
   Ablauf_PO4.Values[114] := 0.0;
   Ablauf_PO4.Values[115] := 0.0;
   Ablauf_PO4.Values[116] := 0.0;
   Ablauf_PO4.Values[117] := 0.0;
   Ablauf_PO4.Values[118] := 0.0;
   Ablauf_PO4.Values[119] := 0.0;
   Umwelt_WG.Values[0] := 0.0;
   Umwelt_WG.Values[1] := 0.0;
   Umwelt_WG.Values[2] := 0.0;
   Umwelt_WG.Values[3] := 0.0;
   Umwelt_WG.Values[4] := 0.0;
   Umwelt_WG.Values[5] := 0.0;
   Umwelt_WG.Values[6] := 0.0;
   Umwelt_WG.Values[7] := 0.0;
   Umwelt_WG.Values[8] := 0.0;
   Umwelt_WG.Values[9] := 0.0;
   Umwelt_WG.Values[10] := 0.0;
   Umwelt_WG.Values[11] := 0.0;
   Umwelt_WG.Values[12] := 0.0;
   Umwelt_WG.Values[13] := 0.0;
   Umwelt_WG.Values[14] := 0.0;
   Umwelt_WG.Values[15] := 0.0;
   Umwelt_WG.Values[16] := 0.0;
   Umwelt_WG.Values[17] := 0.0;
   Umwelt_WG.Values[18] := 0.0;
   Umwelt_WG.Values[19] := 0.0;
   Umwelt_WG.Values[20] := 0.0;
   Umwelt_WG.Values[21] := 0.0;
   Umwelt_WG.Values[22] := 0.0;
   Umwelt_WG.Values[23] := 0.0;
   Umwelt_WG.Values[24] := 0.0;
   Umwelt_WG.Values[25] := 0.0;
   Umwelt_WG.Values[26] := 0.0;
   Umwelt_WG.Values[27] := 0.0;
   Umwelt_WG.Values[28] := 0.0;
   Umwelt_WG.Values[29] := 0.0;
   Umwelt_WG.Values[30] := 0.0;
   Umwelt_WG.Values[31] := 0.0;
   Umwelt_WG.Values[32] := 0.0;
   Umwelt_WG.Values[33] := 0.0;
   Umwelt_WG.Values[34] := 0.0;
   Umwelt_WG.Values[35] := 0.0;
   Umwelt_WG.Values[36] := 0.0;
   Umwelt_WG.Values[37] := 0.0;
   Umwelt_WG.Values[38] := 0.0;
   Umwelt_WG.Values[39] := 0.0;
   Umwelt_WG.Values[40] := 0.0;
   Umwelt_WG.Values[41] := 0.0;
   Umwelt_WG.Values[42] := 0.0;
   Umwelt_WG.Values[43] := 0.0;
   Umwelt_WG.Values[44] := 0.0;
   Umwelt_WG.Values[45] := 0.0;
   Umwelt_WG.Values[46] := 0.0;
   Umwelt_WG.Values[47] := 0.0;
   Umwelt_WG.Values[48] := 0.0;
   Umwelt_WG.Values[49] := 0.0;
   Umwelt_WG.Values[50] := 0.0;
   Umwelt_WG.Values[51] := 0.0;
   Umwelt_WG.Values[52] := 0.0;
   Umwelt_WG.Values[53] := 0.0;
   Umwelt_WG.Values[54] := 0.0;
   Umwelt_WG.Values[55] := 0.0;
   Umwelt_WG.Values[56] := 0.0;
   Umwelt_WG.Values[57] := 0.0;
   Umwelt_WG.Values[58] := 0.0;
   Umwelt_WG.Values[59] := 0.0;
   Umwelt_WG.Values[60] := 0.0;
   Umwelt_WG.Values[61] := 0.0;
   Umwelt_WG.Values[62] := 0.0;
   Umwelt_WG.Values[63] := 0.0;
   Umwelt_WG.Values[64] := 0.0;
   Umwelt_WG.Values[65] := 0.0;
   Umwelt_WG.Values[66] := 0.0;
   Umwelt_WG.Values[67] := 0.0;
   Umwelt_WG.Values[68] := 0.0;
   Umwelt_WG.Values[69] := 0.0;
   Umwelt_WG.Values[70] := 0.0;
   Umwelt_WG.Values[71] := 0.0;
   Umwelt_WG.Values[72] := 0.0;
   Umwelt_WG.Values[73] := 0.0;
   Umwelt_WG.Values[74] := 0.0;
   Umwelt_WG.Values[75] := 0.0;
   Umwelt_WG.Values[76] := 0.0;
   Umwelt_WG.Values[77] := 0.0;
   Umwelt_WG.Values[78] := 0.0;
   Umwelt_WG.Values[79] := 0.0;
   Umwelt_WG.Values[80] := 0.0;
   Umwelt_WG.Values[81] := 0.0;
   Umwelt_WG.Values[82] := 0.0;
   Umwelt_WG.Values[83] := 0.0;
   Umwelt_WG.Values[84] := 0.0;
   Umwelt_WG.Values[85] := 0.0;
   Umwelt_WG.Values[86] := 0.0;
   Umwelt_WG.Values[87] := 0.0;
   Umwelt_WG.Values[88] := 0.0;
   Umwelt_WG.Values[89] := 0.0;
   Umwelt_WG.Values[90] := 0.0;
   Umwelt_WG.Values[91] := 0.0;
   Umwelt_WG.Values[92] := 0.0;
   Umwelt_WG.Values[93] := 0.0;
   Umwelt_WG.Values[94] := 0.0;
   Umwelt_WG.Values[95] := 0.0;
   Umwelt_WG.Values[96] := 0.0;
   Umwelt_WG.Values[97] := 0.0;
   Umwelt_WG.Values[98] := 0.0;
   Umwelt_WG.Values[99] := 0.0;
   Umwelt_WG.Values[100] := 0.0;
   Umwelt_WG.Values[101] := 0.0;
   Umwelt_WG.Values[102] := 0.0;
   Umwelt_WG.Values[103] := 0.0;
   Umwelt_WG.Values[104] := 0.0;
   Umwelt_WG.Values[105] := 0.0;
   Umwelt_WG.Values[106] := 0.0;
   Umwelt_WG.Values[107] := 0.0;
   Umwelt_WG.Values[108] := 0.0;
   Umwelt_WG.Values[109] := 0.0;
   Umwelt_WG.Values[110] := 0.0;
   Umwelt_WG.Values[111] := 0.0;
   Umwelt_WG.Values[112] := 0.0;
   Umwelt_WG.Values[113] := 0.0;
   Umwelt_WG.Values[114] := 0.0;
   Umwelt_WG.Values[115] := 0.0;
   Umwelt_WG.Values[116] := 0.0;
   Umwelt_WG.Values[117] := 0.0;
   Umwelt_WG.Values[118] := 0.0;
   Umwelt_WG.Values[119] := 0.0;
   Umwelt_WR.Values[0] := 0.0;
   Umwelt_WR.Values[1] := 0.0;
   Umwelt_WR.Values[2] := 0.0;
   Umwelt_WR.Values[3] := 0.0;
   Umwelt_WR.Values[4] := 0.0;
   Umwelt_WR.Values[5] := 0.0;
   Umwelt_WR.Values[6] := 0.0;
   Umwelt_WR.Values[7] := 0.0;
   Umwelt_WR.Values[8] := 0.0;
   Umwelt_WR.Values[9] := 0.0;
   Umwelt_WR.Values[10] := 0.0;
   Umwelt_WR.Values[11] := 0.0;
   Umwelt_WR.Values[12] := 0.0;
   Umwelt_WR.Values[13] := 0.0;
   Umwelt_WR.Values[14] := 0.0;
   Umwelt_WR.Values[15] := 0.0;
   Umwelt_WR.Values[16] := 0.0;
   Umwelt_WR.Values[17] := 0.0;
   Umwelt_WR.Values[18] := 0.0;
   Umwelt_WR.Values[19] := 0.0;
   Umwelt_WR.Values[20] := 0.0;
   Umwelt_WR.Values[21] := 0.0;
   Umwelt_WR.Values[22] := 0.0;
   Umwelt_WR.Values[23] := 0.0;
   Umwelt_WR.Values[24] := 0.0;
   Umwelt_WR.Values[25] := 0.0;
   Umwelt_WR.Values[26] := 0.0;
   Umwelt_WR.Values[27] := 0.0;
   Umwelt_WR.Values[28] := 0.0;
   Umwelt_WR.Values[29] := 0.0;
   Umwelt_WR.Values[30] := 0.0;
   Umwelt_WR.Values[31] := 0.0;
   Umwelt_WR.Values[32] := 0.0;
   Umwelt_WR.Values[33] := 0.0;
   Umwelt_WR.Values[34] := 0.0;
   Umwelt_WR.Values[35] := 0.0;
   Umwelt_WR.Values[36] := 0.0;
   Umwelt_WR.Values[37] := 0.0;
   Umwelt_WR.Values[38] := 0.0;
   Umwelt_WR.Values[39] := 0.0;
   Umwelt_WR.Values[40] := 0.0;
   Umwelt_WR.Values[41] := 0.0;
   Umwelt_WR.Values[42] := 0.0;
   Umwelt_WR.Values[43] := 0.0;
   Umwelt_WR.Values[44] := 0.0;
   Umwelt_WR.Values[45] := 0.0;
   Umwelt_WR.Values[46] := 0.0;
   Umwelt_WR.Values[47] := 0.0;
   Umwelt_WR.Values[48] := 0.0;
   Umwelt_WR.Values[49] := 0.0;
   Umwelt_WR.Values[50] := 0.0;
   Umwelt_WR.Values[51] := 0.0;
   Umwelt_WR.Values[52] := 0.0;
   Umwelt_WR.Values[53] := 0.0;
   Umwelt_WR.Values[54] := 0.0;
   Umwelt_WR.Values[55] := 0.0;
   Umwelt_WR.Values[56] := 0.0;
   Umwelt_WR.Values[57] := 0.0;
   Umwelt_WR.Values[58] := 0.0;
   Umwelt_WR.Values[59] := 0.0;
   Umwelt_WR.Values[60] := 0.0;
   Umwelt_WR.Values[61] := 0.0;
   Umwelt_WR.Values[62] := 0.0;
   Umwelt_WR.Values[63] := 0.0;
   Umwelt_WR.Values[64] := 0.0;
   Umwelt_WR.Values[65] := 0.0;
   Umwelt_WR.Values[66] := 0.0;
   Umwelt_WR.Values[67] := 0.0;
   Umwelt_WR.Values[68] := 0.0;
   Umwelt_WR.Values[69] := 0.0;
   Umwelt_WR.Values[70] := 0.0;
   Umwelt_WR.Values[71] := 0.0;
   Umwelt_WR.Values[72] := 0.0;
   Umwelt_WR.Values[73] := 0.0;
   Umwelt_WR.Values[74] := 0.0;
   Umwelt_WR.Values[75] := 0.0;
   Umwelt_WR.Values[76] := 0.0;
   Umwelt_WR.Values[77] := 0.0;
   Umwelt_WR.Values[78] := 0.0;
   Umwelt_WR.Values[79] := 0.0;
   Umwelt_WR.Values[80] := 0.0;
   Umwelt_WR.Values[81] := 0.0;
   Umwelt_WR.Values[82] := 0.0;
   Umwelt_WR.Values[83] := 0.0;
   Umwelt_WR.Values[84] := 0.0;
   Umwelt_WR.Values[85] := 0.0;
   Umwelt_WR.Values[86] := 0.0;
   Umwelt_WR.Values[87] := 0.0;
   Umwelt_WR.Values[88] := 0.0;
   Umwelt_WR.Values[89] := 0.0;
   Umwelt_WR.Values[90] := 0.0;
   Umwelt_WR.Values[91] := 0.0;
   Umwelt_WR.Values[92] := 0.0;
   Umwelt_WR.Values[93] := 0.0;
   Umwelt_WR.Values[94] := 0.0;
   Umwelt_WR.Values[95] := 0.0;
   Umwelt_WR.Values[96] := 0.0;
   Umwelt_WR.Values[97] := 0.0;
   Umwelt_WR.Values[98] := 0.0;
   Umwelt_WR.Values[99] := 0.0;
   Umwelt_WR.Values[100] := 0.0;
   Umwelt_WR.Values[101] := 0.0;
   Umwelt_WR.Values[102] := 0.0;
   Umwelt_WR.Values[103] := 0.0;
   Umwelt_WR.Values[104] := 0.0;
   Umwelt_WR.Values[105] := 0.0;
   Umwelt_WR.Values[106] := 0.0;
   Umwelt_WR.Values[107] := 0.0;
   Umwelt_WR.Values[108] := 0.0;
   Umwelt_WR.Values[109] := 0.0;
   Umwelt_WR.Values[110] := 0.0;
   Umwelt_WR.Values[111] := 0.0;
   Umwelt_WR.Values[112] := 0.0;
   Umwelt_WR.Values[113] := 0.0;
   Umwelt_WR.Values[114] := 0.0;
   Umwelt_WR.Values[115] := 0.0;
   Umwelt_WR.Values[116] := 0.0;
   Umwelt_WR.Values[117] := 0.0;
   Umwelt_WR.Values[118] := 0.0;
   Umwelt_WR.Values[119] := 0.0;
   Umwelt_LDr.Values[0] := 0.0;
   Umwelt_LDr.Values[1] := 0.0;
   Umwelt_LDr.Values[2] := 0.0;
   Umwelt_LDr.Values[3] := 0.0;
   Umwelt_LDr.Values[4] := 0.0;
   Umwelt_LDr.Values[5] := 0.0;
   Umwelt_LDr.Values[6] := 0.0;
   Umwelt_LDr.Values[7] := 0.0;
   Umwelt_LDr.Values[8] := 0.0;
   Umwelt_LDr.Values[9] := 0.0;
   Umwelt_LDr.Values[10] := 0.0;
   Umwelt_LDr.Values[11] := 0.0;
   Umwelt_LDr.Values[12] := 0.0;
   Umwelt_LDr.Values[13] := 0.0;
   Umwelt_LDr.Values[14] := 0.0;
   Umwelt_LDr.Values[15] := 0.0;
   Umwelt_LDr.Values[16] := 0.0;
   Umwelt_LDr.Values[17] := 0.0;
   Umwelt_LDr.Values[18] := 0.0;
   Umwelt_LDr.Values[19] := 0.0;
   Umwelt_LDr.Values[20] := 0.0;
   Umwelt_LDr.Values[21] := 0.0;
   Umwelt_LDr.Values[22] := 0.0;
   Umwelt_LDr.Values[23] := 0.0;
   Umwelt_LDr.Values[24] := 0.0;
   Umwelt_LDr.Values[25] := 0.0;
   Umwelt_LDr.Values[26] := 0.0;
   Umwelt_LDr.Values[27] := 0.0;
   Umwelt_LDr.Values[28] := 0.0;
   Umwelt_LDr.Values[29] := 0.0;
   Umwelt_LDr.Values[30] := 0.0;
   Umwelt_LDr.Values[31] := 0.0;
   Umwelt_LDr.Values[32] := 0.0;
   Umwelt_LDr.Values[33] := 0.0;
   Umwelt_LDr.Values[34] := 0.0;
   Umwelt_LDr.Values[35] := 0.0;
   Umwelt_LDr.Values[36] := 0.0;
   Umwelt_LDr.Values[37] := 0.0;
   Umwelt_LDr.Values[38] := 0.0;
   Umwelt_LDr.Values[39] := 0.0;
   Umwelt_LDr.Values[40] := 0.0;
   Umwelt_LDr.Values[41] := 0.0;
   Umwelt_LDr.Values[42] := 0.0;
   Umwelt_LDr.Values[43] := 0.0;
   Umwelt_LDr.Values[44] := 0.0;
   Umwelt_LDr.Values[45] := 0.0;
   Umwelt_LDr.Values[46] := 0.0;
   Umwelt_LDr.Values[47] := 0.0;
   Umwelt_LDr.Values[48] := 0.0;
   Umwelt_LDr.Values[49] := 0.0;
   Umwelt_LDr.Values[50] := 0.0;
   Umwelt_LDr.Values[51] := 0.0;
   Umwelt_LDr.Values[52] := 0.0;
   Umwelt_LDr.Values[53] := 0.0;
   Umwelt_LDr.Values[54] := 0.0;
   Umwelt_LDr.Values[55] := 0.0;
   Umwelt_LDr.Values[56] := 0.0;
   Umwelt_LDr.Values[57] := 0.0;
   Umwelt_LDr.Values[58] := 0.0;
   Umwelt_LDr.Values[59] := 0.0;
   Umwelt_LDr.Values[60] := 0.0;
   Umwelt_LDr.Values[61] := 0.0;
   Umwelt_LDr.Values[62] := 0.0;
   Umwelt_LDr.Values[63] := 0.0;
   Umwelt_LDr.Values[64] := 0.0;
   Umwelt_LDr.Values[65] := 0.0;
   Umwelt_LDr.Values[66] := 0.0;
   Umwelt_LDr.Values[67] := 0.0;
   Umwelt_LDr.Values[68] := 0.0;
   Umwelt_LDr.Values[69] := 0.0;
   Umwelt_LDr.Values[70] := 0.0;
   Umwelt_LDr.Values[71] := 0.0;
   Umwelt_LDr.Values[72] := 0.0;
   Umwelt_LDr.Values[73] := 0.0;
   Umwelt_LDr.Values[74] := 0.0;
   Umwelt_LDr.Values[75] := 0.0;
   Umwelt_LDr.Values[76] := 0.0;
   Umwelt_LDr.Values[77] := 0.0;
   Umwelt_LDr.Values[78] := 0.0;
   Umwelt_LDr.Values[79] := 0.0;
   Umwelt_LDr.Values[80] := 0.0;
   Umwelt_LDr.Values[81] := 0.0;
   Umwelt_LDr.Values[82] := 0.0;
   Umwelt_LDr.Values[83] := 0.0;
   Umwelt_LDr.Values[84] := 0.0;
   Umwelt_LDr.Values[85] := 0.0;
   Umwelt_LDr.Values[86] := 0.0;
   Umwelt_LDr.Values[87] := 0.0;
   Umwelt_LDr.Values[88] := 0.0;
   Umwelt_LDr.Values[89] := 0.0;
   Umwelt_LDr.Values[90] := 0.0;
   Umwelt_LDr.Values[91] := 0.0;
   Umwelt_LDr.Values[92] := 0.0;
   Umwelt_LDr.Values[93] := 0.0;
   Umwelt_LDr.Values[94] := 0.0;
   Umwelt_LDr.Values[95] := 0.0;
   Umwelt_LDr.Values[96] := 0.0;
   Umwelt_LDr.Values[97] := 0.0;
   Umwelt_LDr.Values[98] := 0.0;
   Umwelt_LDr.Values[99] := 0.0;
   Umwelt_LDr.Values[100] := 0.0;
   Umwelt_LDr.Values[101] := 0.0;
   Umwelt_LDr.Values[102] := 0.0;
   Umwelt_LDr.Values[103] := 0.0;
   Umwelt_LDr.Values[104] := 0.0;
   Umwelt_LDr.Values[105] := 0.0;
   Umwelt_LDr.Values[106] := 0.0;
   Umwelt_LDr.Values[107] := 0.0;
   Umwelt_LDr.Values[108] := 0.0;
   Umwelt_LDr.Values[109] := 0.0;
   Umwelt_LDr.Values[110] := 0.0;
   Umwelt_LDr.Values[111] := 0.0;
   Umwelt_LDr.Values[112] := 0.0;
   Umwelt_LDr.Values[113] := 0.0;
   Umwelt_LDr.Values[114] := 0.0;
   Umwelt_LDr.Values[115] := 0.0;
   Umwelt_LDr.Values[116] := 0.0;
   Umwelt_LDr.Values[117] := 0.0;
   Umwelt_LDr.Values[118] := 0.0;
   Umwelt_LDr.Values[119] := 0.0;
   Umwelt_LF.Values[0] := 0.0;
   Umwelt_LF.Values[1] := 0.0;
   Umwelt_LF.Values[2] := 0.0;
   Umwelt_LF.Values[3] := 0.0;
   Umwelt_LF.Values[4] := 0.0;
   Umwelt_LF.Values[5] := 0.0;
   Umwelt_LF.Values[6] := 0.0;
   Umwelt_LF.Values[7] := 0.0;
   Umwelt_LF.Values[8] := 0.0;
   Umwelt_LF.Values[9] := 0.0;
   Umwelt_LF.Values[10] := 0.0;
   Umwelt_LF.Values[11] := 0.0;
   Umwelt_LF.Values[12] := 0.0;
   Umwelt_LF.Values[13] := 0.0;
   Umwelt_LF.Values[14] := 0.0;
   Umwelt_LF.Values[15] := 0.0;
   Umwelt_LF.Values[16] := 0.0;
   Umwelt_LF.Values[17] := 0.0;
   Umwelt_LF.Values[18] := 0.0;
   Umwelt_LF.Values[19] := 0.0;
   Umwelt_LF.Values[20] := 0.0;
   Umwelt_LF.Values[21] := 0.0;
   Umwelt_LF.Values[22] := 0.0;
   Umwelt_LF.Values[23] := 0.0;
   Umwelt_LF.Values[24] := 0.0;
   Umwelt_LF.Values[25] := 0.0;
   Umwelt_LF.Values[26] := 0.0;
   Umwelt_LF.Values[27] := 0.0;
   Umwelt_LF.Values[28] := 0.0;
   Umwelt_LF.Values[29] := 0.0;
   Umwelt_LF.Values[30] := 0.0;
   Umwelt_LF.Values[31] := 0.0;
   Umwelt_LF.Values[32] := 0.0;
   Umwelt_LF.Values[33] := 0.0;
   Umwelt_LF.Values[34] := 0.0;
   Umwelt_LF.Values[35] := 0.0;
   Umwelt_LF.Values[36] := 0.0;
   Umwelt_LF.Values[37] := 0.0;
   Umwelt_LF.Values[38] := 0.0;
   Umwelt_LF.Values[39] := 0.0;
   Umwelt_LF.Values[40] := 0.0;
   Umwelt_LF.Values[41] := 0.0;
   Umwelt_LF.Values[42] := 0.0;
   Umwelt_LF.Values[43] := 0.0;
   Umwelt_LF.Values[44] := 0.0;
   Umwelt_LF.Values[45] := 0.0;
   Umwelt_LF.Values[46] := 0.0;
   Umwelt_LF.Values[47] := 0.0;
   Umwelt_LF.Values[48] := 0.0;
   Umwelt_LF.Values[49] := 0.0;
   Umwelt_LF.Values[50] := 0.0;
   Umwelt_LF.Values[51] := 0.0;
   Umwelt_LF.Values[52] := 0.0;
   Umwelt_LF.Values[53] := 0.0;
   Umwelt_LF.Values[54] := 0.0;
   Umwelt_LF.Values[55] := 0.0;
   Umwelt_LF.Values[56] := 0.0;
   Umwelt_LF.Values[57] := 0.0;
   Umwelt_LF.Values[58] := 0.0;
   Umwelt_LF.Values[59] := 0.0;
   Umwelt_LF.Values[60] := 0.0;
   Umwelt_LF.Values[61] := 0.0;
   Umwelt_LF.Values[62] := 0.0;
   Umwelt_LF.Values[63] := 0.0;
   Umwelt_LF.Values[64] := 0.0;
   Umwelt_LF.Values[65] := 0.0;
   Umwelt_LF.Values[66] := 0.0;
   Umwelt_LF.Values[67] := 0.0;
   Umwelt_LF.Values[68] := 0.0;
   Umwelt_LF.Values[69] := 0.0;
   Umwelt_LF.Values[70] := 0.0;
   Umwelt_LF.Values[71] := 0.0;
   Umwelt_LF.Values[72] := 0.0;
   Umwelt_LF.Values[73] := 0.0;
   Umwelt_LF.Values[74] := 0.0;
   Umwelt_LF.Values[75] := 0.0;
   Umwelt_LF.Values[76] := 0.0;
   Umwelt_LF.Values[77] := 0.0;
   Umwelt_LF.Values[78] := 0.0;
   Umwelt_LF.Values[79] := 0.0;
   Umwelt_LF.Values[80] := 0.0;
   Umwelt_LF.Values[81] := 0.0;
   Umwelt_LF.Values[82] := 0.0;
   Umwelt_LF.Values[83] := 0.0;
   Umwelt_LF.Values[84] := 0.0;
   Umwelt_LF.Values[85] := 0.0;
   Umwelt_LF.Values[86] := 0.0;
   Umwelt_LF.Values[87] := 0.0;
   Umwelt_LF.Values[88] := 0.0;
   Umwelt_LF.Values[89] := 0.0;
   Umwelt_LF.Values[90] := 0.0;
   Umwelt_LF.Values[91] := 0.0;
   Umwelt_LF.Values[92] := 0.0;
   Umwelt_LF.Values[93] := 0.0;
   Umwelt_LF.Values[94] := 0.0;
   Umwelt_LF.Values[95] := 0.0;
   Umwelt_LF.Values[96] := 0.0;
   Umwelt_LF.Values[97] := 0.0;
   Umwelt_LF.Values[98] := 0.0;
   Umwelt_LF.Values[99] := 0.0;
   Umwelt_LF.Values[100] := 0.0;
   Umwelt_LF.Values[101] := 0.0;
   Umwelt_LF.Values[102] := 0.0;
   Umwelt_LF.Values[103] := 0.0;
   Umwelt_LF.Values[104] := 0.0;
   Umwelt_LF.Values[105] := 0.0;
   Umwelt_LF.Values[106] := 0.0;
   Umwelt_LF.Values[107] := 0.0;
   Umwelt_LF.Values[108] := 0.0;
   Umwelt_LF.Values[109] := 0.0;
   Umwelt_LF.Values[110] := 0.0;
   Umwelt_LF.Values[111] := 0.0;
   Umwelt_LF.Values[112] := 0.0;
   Umwelt_LF.Values[113] := 0.0;
   Umwelt_LF.Values[114] := 0.0;
   Umwelt_LF.Values[115] := 0.0;
   Umwelt_LF.Values[116] := 0.0;
   Umwelt_LF.Values[117] := 0.0;
   Umwelt_LF.Values[118] := 0.0;
   Umwelt_LF.Values[119] := 0.0;
   Umwelt_T.Values[0] := 0.0;
   Umwelt_T.Values[1] := 0.0;
   Umwelt_T.Values[2] := 0.0;
   Umwelt_T.Values[3] := 0.0;
   Umwelt_T.Values[4] := 0.0;
   Umwelt_T.Values[5] := 0.0;
   Umwelt_T.Values[6] := 0.0;
   Umwelt_T.Values[7] := 0.0;
   Umwelt_T.Values[8] := 0.0;
   Umwelt_T.Values[9] := 0.0;
   Umwelt_T.Values[10] := 0.0;
   Umwelt_T.Values[11] := 0.0;
   Umwelt_T.Values[12] := 0.0;
   Umwelt_T.Values[13] := 0.0;
   Umwelt_T.Values[14] := 0.0;
   Umwelt_T.Values[15] := 0.0;
   Umwelt_T.Values[16] := 0.0;
   Umwelt_T.Values[17] := 0.0;
   Umwelt_T.Values[18] := 0.0;
   Umwelt_T.Values[19] := 0.0;
   Umwelt_T.Values[20] := 0.0;
   Umwelt_T.Values[21] := 0.0;
   Umwelt_T.Values[22] := 0.0;
   Umwelt_T.Values[23] := 0.0;
   Umwelt_T.Values[24] := 0.0;
   Umwelt_T.Values[25] := 0.0;
   Umwelt_T.Values[26] := 0.0;
   Umwelt_T.Values[27] := 0.0;
   Umwelt_T.Values[28] := 0.0;
   Umwelt_T.Values[29] := 0.0;
   Umwelt_T.Values[30] := 0.0;
   Umwelt_T.Values[31] := 0.0;
   Umwelt_T.Values[32] := 0.0;
   Umwelt_T.Values[33] := 0.0;
   Umwelt_T.Values[34] := 0.0;
   Umwelt_T.Values[35] := 0.0;
   Umwelt_T.Values[36] := 0.0;
   Umwelt_T.Values[37] := 0.0;
   Umwelt_T.Values[38] := 0.0;
   Umwelt_T.Values[39] := 0.0;
   Umwelt_T.Values[40] := 0.0;
   Umwelt_T.Values[41] := 0.0;
   Umwelt_T.Values[42] := 0.0;
   Umwelt_T.Values[43] := 0.0;
   Umwelt_T.Values[44] := 0.0;
   Umwelt_T.Values[45] := 0.0;
   Umwelt_T.Values[46] := 0.0;
   Umwelt_T.Values[47] := 0.0;
   Umwelt_T.Values[48] := 0.0;
   Umwelt_T.Values[49] := 0.0;
   Umwelt_T.Values[50] := 0.0;
   Umwelt_T.Values[51] := 0.0;
   Umwelt_T.Values[52] := 0.0;
   Umwelt_T.Values[53] := 0.0;
   Umwelt_T.Values[54] := 0.0;
   Umwelt_T.Values[55] := 0.0;
   Umwelt_T.Values[56] := 0.0;
   Umwelt_T.Values[57] := 0.0;
   Umwelt_T.Values[58] := 0.0;
   Umwelt_T.Values[59] := 0.0;
   Umwelt_T.Values[60] := 0.0;
   Umwelt_T.Values[61] := 0.0;
   Umwelt_T.Values[62] := 0.0;
   Umwelt_T.Values[63] := 0.0;
   Umwelt_T.Values[64] := 0.0;
   Umwelt_T.Values[65] := 0.0;
   Umwelt_T.Values[66] := 0.0;
   Umwelt_T.Values[67] := 0.0;
   Umwelt_T.Values[68] := 0.0;
   Umwelt_T.Values[69] := 0.0;
   Umwelt_T.Values[70] := 0.0;
   Umwelt_T.Values[71] := 0.0;
   Umwelt_T.Values[72] := 0.0;
   Umwelt_T.Values[73] := 0.0;
   Umwelt_T.Values[74] := 0.0;
   Umwelt_T.Values[75] := 0.0;
   Umwelt_T.Values[76] := 0.0;
   Umwelt_T.Values[77] := 0.0;
   Umwelt_T.Values[78] := 0.0;
   Umwelt_T.Values[79] := 0.0;
   Umwelt_T.Values[80] := 0.0;
   Umwelt_T.Values[81] := 0.0;
   Umwelt_T.Values[82] := 0.0;
   Umwelt_T.Values[83] := 0.0;
   Umwelt_T.Values[84] := 0.0;
   Umwelt_T.Values[85] := 0.0;
   Umwelt_T.Values[86] := 0.0;
   Umwelt_T.Values[87] := 0.0;
   Umwelt_T.Values[88] := 0.0;
   Umwelt_T.Values[89] := 0.0;
   Umwelt_T.Values[90] := 0.0;
   Umwelt_T.Values[91] := 0.0;
   Umwelt_T.Values[92] := 0.0;
   Umwelt_T.Values[93] := 0.0;
   Umwelt_T.Values[94] := 0.0;
   Umwelt_T.Values[95] := 0.0;
   Umwelt_T.Values[96] := 0.0;
   Umwelt_T.Values[97] := 0.0;
   Umwelt_T.Values[98] := 0.0;
   Umwelt_T.Values[99] := 0.0;
   Umwelt_T.Values[100] := 0.0;
   Umwelt_T.Values[101] := 0.0;
   Umwelt_T.Values[102] := 0.0;
   Umwelt_T.Values[103] := 0.0;
   Umwelt_T.Values[104] := 0.0;
   Umwelt_T.Values[105] := 0.0;
   Umwelt_T.Values[106] := 0.0;
   Umwelt_T.Values[107] := 0.0;
   Umwelt_T.Values[108] := 0.0;
   Umwelt_T.Values[109] := 0.0;
   Umwelt_T.Values[110] := 0.0;
   Umwelt_T.Values[111] := 0.0;
   Umwelt_T.Values[112] := 0.0;
   Umwelt_T.Values[113] := 0.0;
   Umwelt_T.Values[114] := 0.0;
   Umwelt_T.Values[115] := 0.0;
   Umwelt_T.Values[116] := 0.0;
   Umwelt_T.Values[117] := 0.0;
   Umwelt_T.Values[118] := 0.0;
   Umwelt_T.Values[119] := 0.0;
   Ablauf_LF.Values[0] := 0.0;
   Ablauf_LF.Values[1] := 0.0;
   Ablauf_LF.Values[2] := 0.0;
   Ablauf_LF.Values[3] := 0.0;
   Ablauf_LF.Values[4] := 0.0;
   Ablauf_LF.Values[5] := 0.0;
   Ablauf_LF.Values[6] := 0.0;
   Ablauf_LF.Values[7] := 0.0;
   Ablauf_LF.Values[8] := 0.0;
   Ablauf_LF.Values[9] := 0.0;
   Ablauf_LF.Values[10] := 0.0;
   Ablauf_LF.Values[11] := 0.0;
   Ablauf_LF.Values[12] := 0.0;
   Ablauf_LF.Values[13] := 0.0;
   Ablauf_LF.Values[14] := 0.0;
   Ablauf_LF.Values[15] := 0.0;
   Ablauf_LF.Values[16] := 0.0;
   Ablauf_LF.Values[17] := 0.0;
   Ablauf_LF.Values[18] := 0.0;
   Ablauf_LF.Values[19] := 0.0;
   Ablauf_LF.Values[20] := 0.0;
   Ablauf_LF.Values[21] := 0.0;
   Ablauf_LF.Values[22] := 0.0;
   Ablauf_LF.Values[23] := 0.0;
   Ablauf_LF.Values[24] := 0.0;
   Ablauf_LF.Values[25] := 0.0;
   Ablauf_LF.Values[26] := 0.0;
   Ablauf_LF.Values[27] := 0.0;
   Ablauf_LF.Values[28] := 0.0;
   Ablauf_LF.Values[29] := 0.0;
   Ablauf_LF.Values[30] := 0.0;
   Ablauf_LF.Values[31] := 0.0;
   Ablauf_LF.Values[32] := 0.0;
   Ablauf_LF.Values[33] := 0.0;
   Ablauf_LF.Values[34] := 0.0;
   Ablauf_LF.Values[35] := 0.0;
   Ablauf_LF.Values[36] := 0.0;
   Ablauf_LF.Values[37] := 0.0;
   Ablauf_LF.Values[38] := 0.0;
   Ablauf_LF.Values[39] := 0.0;
   Ablauf_LF.Values[40] := 0.0;
   Ablauf_LF.Values[41] := 0.0;
   Ablauf_LF.Values[42] := 0.0;
   Ablauf_LF.Values[43] := 0.0;
   Ablauf_LF.Values[44] := 0.0;
   Ablauf_LF.Values[45] := 0.0;
   Ablauf_LF.Values[46] := 0.0;
   Ablauf_LF.Values[47] := 0.0;
   Ablauf_LF.Values[48] := 0.0;
   Ablauf_LF.Values[49] := 0.0;
   Ablauf_LF.Values[50] := 0.0;
   Ablauf_LF.Values[51] := 0.0;
   Ablauf_LF.Values[52] := 0.0;
   Ablauf_LF.Values[53] := 0.0;
   Ablauf_LF.Values[54] := 0.0;
   Ablauf_LF.Values[55] := 0.0;
   Ablauf_LF.Values[56] := 0.0;
   Ablauf_LF.Values[57] := 0.0;
   Ablauf_LF.Values[58] := 0.0;
   Ablauf_LF.Values[59] := 0.0;
   Ablauf_LF.Values[60] := 0.0;
   Ablauf_LF.Values[61] := 0.0;
   Ablauf_LF.Values[62] := 0.0;
   Ablauf_LF.Values[63] := 0.0;
   Ablauf_LF.Values[64] := 0.0;
   Ablauf_LF.Values[65] := 0.0;
   Ablauf_LF.Values[66] := 0.0;
   Ablauf_LF.Values[67] := 0.0;
   Ablauf_LF.Values[68] := 0.0;
   Ablauf_LF.Values[69] := 0.0;
   Ablauf_LF.Values[70] := 0.0;
   Ablauf_LF.Values[71] := 0.0;
   Ablauf_LF.Values[72] := 0.0;
   Ablauf_LF.Values[73] := 0.0;
   Ablauf_LF.Values[74] := 0.0;
   Ablauf_LF.Values[75] := 0.0;
   Ablauf_LF.Values[76] := 0.0;
   Ablauf_LF.Values[77] := 0.0;
   Ablauf_LF.Values[78] := 0.0;
   Ablauf_LF.Values[79] := 0.0;
   Ablauf_LF.Values[80] := 0.0;
   Ablauf_LF.Values[81] := 0.0;
   Ablauf_LF.Values[82] := 0.0;
   Ablauf_LF.Values[83] := 0.0;
   Ablauf_LF.Values[84] := 0.0;
   Ablauf_LF.Values[85] := 0.0;
   Ablauf_LF.Values[86] := 0.0;
   Ablauf_LF.Values[87] := 0.0;
   Ablauf_LF.Values[88] := 0.0;
   Ablauf_LF.Values[89] := 0.0;
   Ablauf_LF.Values[90] := 0.0;
   Ablauf_LF.Values[91] := 0.0;
   Ablauf_LF.Values[92] := 0.0;
   Ablauf_LF.Values[93] := 0.0;
   Ablauf_LF.Values[94] := 0.0;
   Ablauf_LF.Values[95] := 0.0;
   Ablauf_LF.Values[96] := 0.0;
   Ablauf_LF.Values[97] := 0.0;
   Ablauf_LF.Values[98] := 0.0;
   Ablauf_LF.Values[99] := 0.0;
   Ablauf_LF.Values[100] := 0.0;
   Ablauf_LF.Values[101] := 0.0;
   Ablauf_LF.Values[102] := 0.0;
   Ablauf_LF.Values[103] := 0.0;
   Ablauf_LF.Values[104] := 0.0;
   Ablauf_LF.Values[105] := 0.0;
   Ablauf_LF.Values[106] := 0.0;
   Ablauf_LF.Values[107] := 0.0;
   Ablauf_LF.Values[108] := 0.0;
   Ablauf_LF.Values[109] := 0.0;
   Ablauf_LF.Values[110] := 0.0;
   Ablauf_LF.Values[111] := 0.0;
   Ablauf_LF.Values[112] := 0.0;
   Ablauf_LF.Values[113] := 0.0;
   Ablauf_LF.Values[114] := 0.0;
   Ablauf_LF.Values[115] := 0.0;
   Ablauf_LF.Values[116] := 0.0;
   Ablauf_LF.Values[117] := 0.0;
   Ablauf_LF.Values[118] := 0.0;
   Ablauf_LF.Values[119] := 0.0;

END_DATA_BLOCK

DATA_BLOCK "DB96_ZW"
{ S7_Optimized_Access := 'FALSE' }
VERSION : 0.1
   STRUCT
      Zulauf_AR_DF { ExternalAccessible := 'False'; ExternalVisible := 'False'; ExternalWritable := 'False'} : "T_ZW_BEF";
      BB1_DF { ExternalAccessible := 'False'; ExternalVisible := 'False'; ExternalWritable := 'False'} : "T_ZW_BEF";
      BB2_DF { ExternalAccessible := 'False'; ExternalVisible := 'False'; ExternalWritable := 'False'} : "T_ZW_BEF";
      Zulauf_DF { ExternalAccessible := 'False'; ExternalVisible := 'False'; ExternalWritable := 'False'} : "T_ZW_BEF";
      BB_UeSS_DF { ExternalAccessible := 'False'; ExternalVisible := 'False'; ExternalWritable := 'False'} : "T_ZW_BEF";
      Ablauf_DF { ExternalAccessible := 'False'; ExternalVisible := 'False'; ExternalWritable := 'False'} : "T_ZW_BEF";
      Schlamm_Besch_DF { ExternalAccessible := 'False'; ExternalVisible := 'False'; ExternalWritable := 'False'} : "T_ZW_BEF";
      Truebwasser_DF { ExternalAccessible := 'False'; ExternalVisible := 'False'; ExternalWritable := 'False'} : "T_ZW_BEF";
      BB_Biocos_DF { ExternalAccessible := 'False'; ExternalVisible := 'False'; ExternalWritable := 'False'} : "T_ZW_BEF";
      Umwelt_RM { ExternalAccessible := 'False'; ExternalVisible := 'False'; ExternalWritable := 'False'} : "T_ZW_BEF";   // Regenmenge in 0,1 mm
   END_STRUCT;


BEGIN
   Zulauf_AR_DF.Reset := FALSE;
   Zulauf_AR_DF.Impuls := FALSE;
   Zulauf_AR_DF.Teiler := 1;
   Zulauf_AR_DF.ZW_raw := 583302;
   Zulauf_AR_DF.ZW_Tag := 0;
   Zulauf_AR_DF.ZW_Vortag := 0;
   BB1_DF.Reset := FALSE;
   BB1_DF.Impuls := FALSE;
   BB1_DF.Teiler := 1;
   BB1_DF.ZW_raw := 0;
   BB1_DF.ZW_Tag := 0;
   BB1_DF.ZW_Vortag := 0;
   BB2_DF.Reset := FALSE;
   BB2_DF.Impuls := FALSE;
   BB2_DF.Teiler := 1;
   BB2_DF.ZW_raw := 0;
   BB2_DF.ZW_Tag := 0;
   BB2_DF.ZW_Vortag := 0;
   Zulauf_DF.Reset := FALSE;
   Zulauf_DF.Impuls := FALSE;
   Zulauf_DF.Teiler := 1;
   Zulauf_DF.ZW_raw := 1741323;
   Zulauf_DF.ZW_Tag := 1066;
   Zulauf_DF.ZW_Vortag := 905;
   BB_UeSS_DF.Reset := FALSE;
   BB_UeSS_DF.Impuls := FALSE;
   BB_UeSS_DF.Teiler := 1;
   BB_UeSS_DF.ZW_raw := 821774;
   BB_UeSS_DF.ZW_Tag := 390;
   BB_UeSS_DF.ZW_Vortag := 390;
   Ablauf_DF.Reset := FALSE;
   Ablauf_DF.Impuls := FALSE;
   Ablauf_DF.Teiler := 1;
   Ablauf_DF.ZW_raw := 1542274;
   Ablauf_DF.ZW_Tag := 869;
   Ablauf_DF.ZW_Vortag := 815;
   Schlamm_Besch_DF.Reset := FALSE;
   Schlamm_Besch_DF.Impuls := FALSE;
   Schlamm_Besch_DF.Teiler := 1;
   Schlamm_Besch_DF.ZW_raw := 53300;
   Schlamm_Besch_DF.ZW_Tag := 0;
   Schlamm_Besch_DF.ZW_Vortag := 0;
   Truebwasser_DF.Reset := FALSE;
   Truebwasser_DF.Impuls := FALSE;
   Truebwasser_DF.Teiler := 1;
   Truebwasser_DF.ZW_raw := 207644;
   Truebwasser_DF.ZW_Tag := 89;
   Truebwasser_DF.ZW_Vortag := 90;
   BB_Biocos_DF.Reset := FALSE;
   BB_Biocos_DF.Impuls := FALSE;
   BB_Biocos_DF.Teiler := 1;
   BB_Biocos_DF.ZW_raw := 0;
   BB_Biocos_DF.ZW_Tag := 0;
   BB_Biocos_DF.ZW_Vortag := 0;

END_DATA_BLOCK

DATA_BLOCK "ZEN_EA"
{ S7_Optimized_Access := 'FALSE' }
VERSION : 0.1
NON_RETAIN
   STRUCT
      EW_Zulauf_AR_Niv : Word;   // Zulauf - Pumpwerk "Alter Rechen" - Niveau - Messwert von analoger Peripherie
      EW_Zulauf_AR_Temp : Word;   // Zulauf - Pumpwerk "Alter Rechen" - Temperatur - Messwert von analoger Peripherie
      EW_Zulauf_AR_DF : Word;   // Zulauf - Pumpwerk "Alter Rechen" - Durchfluss - Messwert von analoger Peripherie
      EW_Ablauf_DF : Word;   // Ablauf - Durchfluss - Messwert von analoger Peripherie
      EW_Ablauf_pH : Word;   // Ablauf - pH-Wert - Messwert von analoger Peripherie
      EW_Ablauf_O2 : Word;   // Ablauf - O2-Gehalt - Messwert von analoger Peripherie
      EW_Ablauf_Temp : Word;   // Ablauf - Temperatur - Messwert von analoger Peripherie
      EW_BB_UeSS_DF : Word;   // Becken 1+2 - Ablauf ÜSS - Durchfluss - Messwert von analoger Peripherie
      EW_ZEN_Res_320 : Word;   // Reserve
      EW_ZEN_Res_322 : Word;   // Reserve
      EW_ZEN_Res_324 : Word;   // Reserve
      EW_ZEN_Res_326 : Word;   // Reserve
      EW_ZEN_Res_328 : Word;   // Reserve
      EW_ZEN_Res_330 : Word;   // Reserve
      EW_ZEN_Res_332 : Word;   // Reserve
      EW_ZEN_Res_334 : Word;   // Reserve
      EW_BB1_AS1_SS : Word;   // Becken 1 - Ablaufschieber 1 - Schieberstellung - Messwert von analoger Peripherie
      EW_BB1_AS2_SS : Word;   // Becken 1 - Ablaufschieber 2 - Schieberstellung - Messwert von analoger Peripherie
      EW_BB2_AS1_SS : Word;   // Becken 2 - Ablaufschieber 1 - Schieberstellung - Messwert von analoger Peripherie
      EW_BB2_AS2_SS : Word;   // Becken 2 - Ablaufschieber 2 - Schieberstellung - Messwert von analoger Peripherie
      EW_BB1_O2 : Word;   // Becken 1 - O2-Gehalt - Messwert von analoger Peripherie
      EW_BB1_Temp : Word;   // Becken 1 - Temperatur - Messwert von analoger Peripherie
      EW_BB2_O2 : Word;   // Becken 2 - O2-Gehalt - Messwert von analoger Peripherie
      EW_BB2_Temp : Word;   // Becken 2 - Temperatur - Messwert von analoger Peripherie
      EW_BB1_DF : Word;   // Becken 1 - Ablauf - Durchfluss - Messwert von analoger Peripherie
      EW_BB2_DF : Word;   // Becken 2 - Ablauf - Durchfluss - Messwert von analoger Peripherie
      EW_Zulauf_Niv : Word;   // Zulauf - Vorlagebehälter - Niveau - Messwert von analoger Peripherie
      EW_Zulauf_DF : Word;   // Zulauf - Rechen - Durchfluss - Messwert von analoger Peripherie
      EW_Verteiler_pH : Word;   // Zulauf - Verteiler - pH-Wert - Messwert von analoger Peripherie
      EW_Verteiler_O2 : Word;   // Zulauf - Verteiler  - O2-Gehalt - Messwert von analoger Peripherie
      EW_Zulauf_SF_Niv : Word;   // Zulauf - Sandfang - Niveau - Messwert von analoger Peripherie
      EW_Verteiler_Temp : Word;   // Zulauf - Verteiler - Temperatur - Messwert von analoger Peripherie
      EW_Schlamm_Besch_DF : Word;   // Schlamm - Beschickung - Durchfluss - Messwert von analoger Peripherie
      EW_Truebwasser_Niv : Word;   // Trübwasserpumpwerk - Niveau - Messwert von analoger Peripherie
      EW_Truebwasser_DF : Word;   // Trübwasserpumpwerk - Durchfluss - Messwert von analoger Peripherie
      EW_ZEN_Res_310 : Word;   // Reserve
      EW_ZEN_Res_312 : Word;   // Reserve
      EW_ZEN_Res_314 : Word;   // Reserve
      EW_ZEN_Res_316 : Word;   // Reserve
      EW_ZEN_Res_318 : Word;   // Reserve
      EW_Umwelt_WG : Word;   // Wetterstation - Windgeschwindigkeit
      EW_Umwelt_WR : Word;   // Wetterstation - Windrichtung
      EW_Umwelt_LDr : Word;   // Wetterstation - Luftdruck
      EW_Umwelt_LF : Word;   // Wetterstation - Luftfeuchtigkeit
      EW_Umwelt_T : Word;   // Wetterstation - Temperatur
      EW_Ablauf_LF : Word;   // Ablauf - Leitfähigkeit
      EW_ZEN_Res_404 : Word;   // Reserve
      EW_ZEN_Res_406 : Word;   // Reserve
      RES : Array[0..9] of Byte;
   END_STRUCT;


BEGIN

END_DATA_BLOCK

DATA_BLOCK "FB7_Pumpwerke_IDB"
{ S7_Optimized_Access := 'FALSE' }
VERSION : 0.1
NON_RETAIN
"FB7_Pumpwerke"

BEGIN

END_DATA_BLOCK

DATA_BLOCK "FB9_USV_Kom_IDB"
{ S7_Optimized_Access := 'TRUE' }
VERSION : 0.1
NON_RETAIN
"FB9_USV_Kom"

BEGIN

END_DATA_BLOCK

DATA_BLOCK "FB8_Leitstelle_IDB"
{ S7_Optimized_Access := 'TRUE' }
VERSION : 0.1
NON_RETAIN
"FB8_Leitstelle"

BEGIN

END_DATA_BLOCK

DATA_BLOCK "FB1_Antriebe_IDB"
{ S7_Optimized_Access := 'TRUE' }
VERSION : 0.1
NON_RETAIN
"FB1_Antriebe"

